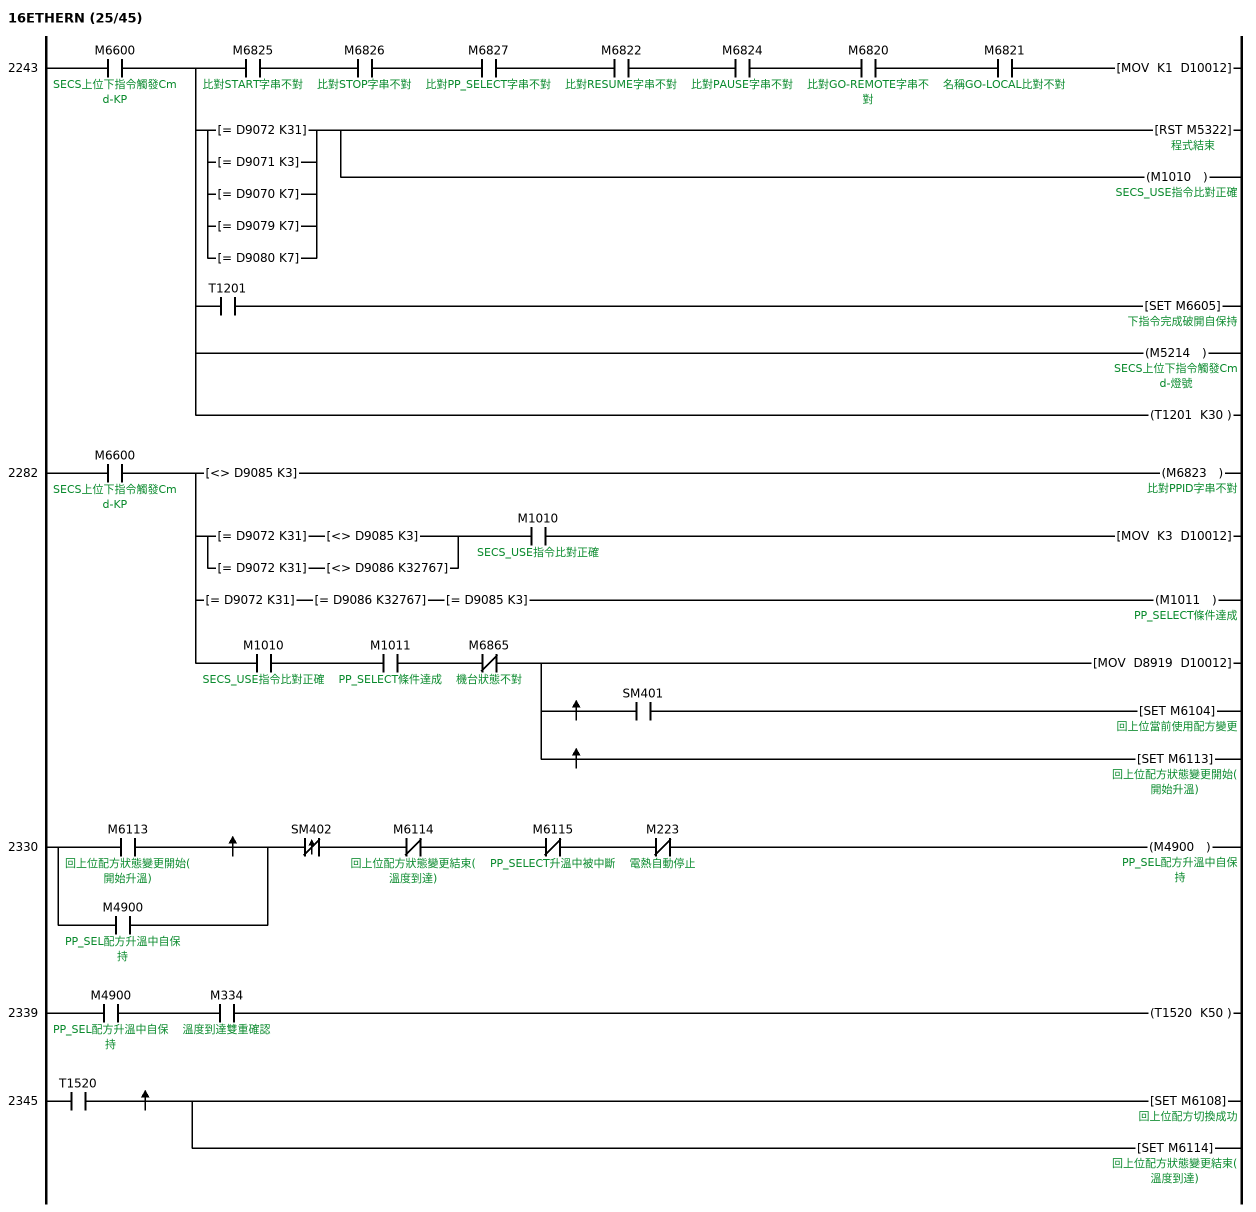
[picture p120: ladder of 16ETHERN, rungs at steps 2243 to 2345]
2243  LD      M6600  ; SECS上位下指令觸發Cmd-KP
      MPS
      AND     M6825  ; 比對START字串不對
      AND     M6826  ; 比對STOP字串不對
      AND     M6827  ; 比對PP_SELECT字串不對
      AND     M6822  ; 比對RESUME字串不對
      AND     M6824  ; 比對PAUSE字串不對
      AND     M6820  ; 比對GO-REMOTE字串不對
      AND     M6821  ; 名稱GO-LOCAL比對不對
      MOV     K1 D10012
      MRD
      LD=     D9072 K31
      OR=     D9071 K3
      OR=     D9070 K7
      OR=     D9079 K7
      OR=     D9080 K7
      ANB
      RST     M5322  ; 程式結束
      OUT     M1010  ; SECS_USE指令比對正確
      MRD
      AND     T1201
      SET     M6605  ; 下指令完成破開自保持
      MPP
      OUT     M5214  ; SECS上位下指令觸發Cmd-燈號
      OUT     T1201 K30
2282  LD      M6600  ; SECS上位下指令觸發Cmd-KP
      MPS
      AND<>   D9085 K3
      OUT     M6823  ; 比對PPID字串不對
      MRD
      LD=     D9072 K31
      AND<>   D9085 K3
      LD=     D9072 K31
      AND<>   D9086 K32767
      ORB
      ANB
      AND     M1010  ; SECS_USE指令比對正確
      MOV     K3 D10012
      MRD
      AND=    D9072 K31
      AND=    D9086 K32767
      AND=    D9085 K3
      OUT     M1011  ; PP_SELECT條件達成
      MPP
      AND     M1010  ; SECS_USE指令比對正確
      AND     M1011  ; PP_SELECT條件達成
      ANI     M6865  ; 機台狀態不對
      MOV     D8919 D10012
      MPS
      MEP
      AND     SM401
      SET     M6104  ; 回上位當前使用配方變更
      MPP
      MEP
      SET     M6113  ; 回上位配方狀態變更開始(開始升溫)
2330  LD      M6113  ; 回上位配方狀態變更開始(開始升溫)
      MEP
      OR      M4900  ; PP_SEL配方升溫中自保持
      ANDPI   SM402
      ANI     M6114  ; 回上位配方狀態變更結束(溫度到達)
      ANI     M6115  ; PP_SELECT升溫中被中斷
      ANI     M223  ; 電熱自動停止
      OUT     M4900  ; PP_SEL配方升溫中自保持
2339  LD      M4900  ; PP_SEL配方升溫中自保持
      AND     M334  ; 溫度到達雙重確認
      OUT     T1520 K50
2345  LD      T1520
      MEP
      SET     M6108  ; 回上位配方切換成功
      SET     M6114  ; 回上位配方狀態變更結束(溫度到達)
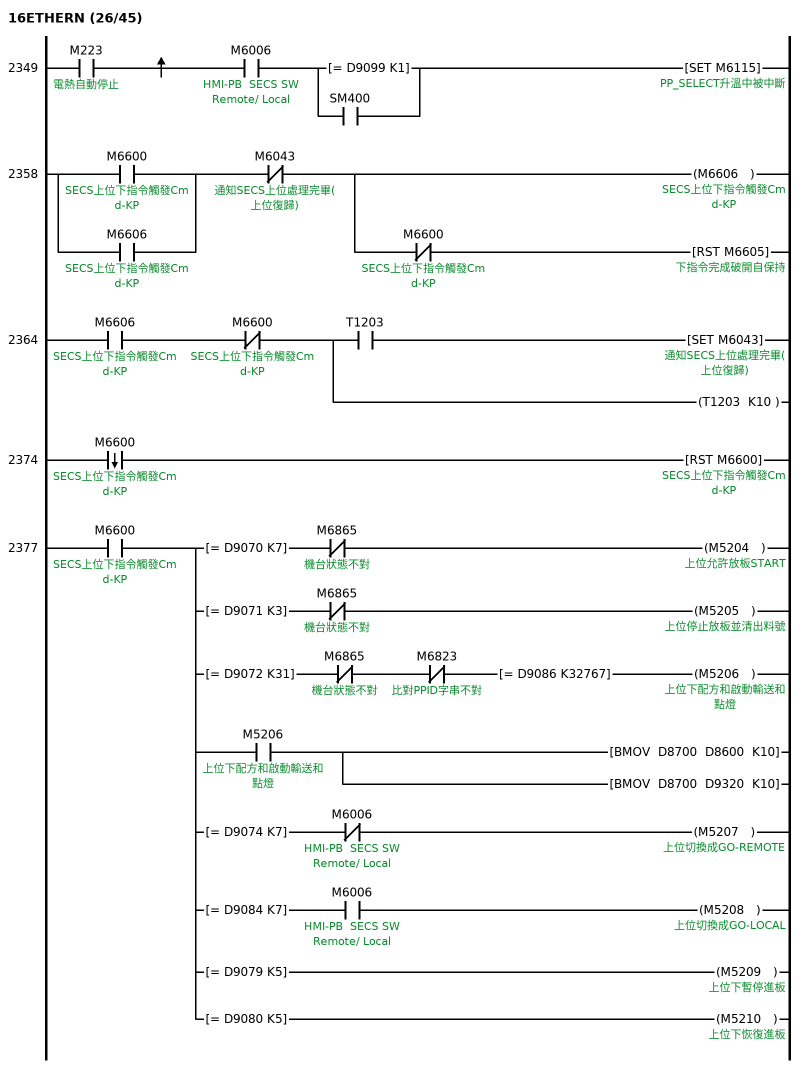
2349  LD      M223  ; 電熱自動停止
      MEP
      AND     M6006  ; HMI-PB  SECS SW  Remote/ Local
      LD=     D9099 K1
      OR      SM400
      ANB
      SET     M6115  ; PP_SELECT升溫中被中斷
2358  LD      M6600  ; SECS上位下指令觸發Cmd-KP
      OR      M6606  ; SECS上位下指令觸發Cmd-KP
      ANI     M6043  ; 通知SECS上位處理完畢(上位復歸)
      OUT     M6606  ; SECS上位下指令觸發Cmd-KP
      ANI     M6600  ; SECS上位下指令觸發Cmd-KP
      RST     M6605  ; 下指令完成破開自保持
2364  LD      M6606  ; SECS上位下指令觸發Cmd-KP
      ANI     M6600  ; SECS上位下指令觸發Cmd-KP
      MPS
      AND     T1203
      SET     M6043  ; 通知SECS上位處理完畢(上位復歸)
      MPP
      OUT     T1203 K10
2374  LDF     M6600  ; SECS上位下指令觸發Cmd-KP
      RST     M6600  ; SECS上位下指令觸發Cmd-KP
2377  LD      M6600  ; SECS上位下指令觸發Cmd-KP
      MPS
      AND=    D9070 K7
      ANI     M6865  ; 機台狀態不對
      OUT     M5204  ; 上位允許放板START
      MRD
      AND=    D9071 K3
      ANI     M6865  ; 機台狀態不對
      OUT     M5205  ; 上位停止放板並清出料號
      MRD
      AND=    D9072 K31
      ANI     M6865  ; 機台狀態不對
      ANI     M6823  ; 比對PPID字串不對
      AND=    D9086 K32767
      OUT     M5206  ; 上位下配方和啟動輸送和點燈
      MRD
      AND     M5206  ; 上位下配方和啟動輸送和點燈
      BMOV    D8700 D8600 K10
      BMOV    D8700 D9320 K10
      MRD
      AND=    D9074 K7
      ANI     M6006  ; HMI-PB  SECS SW  Remote/ Local
      OUT     M5207  ; 上位切換成GO-REMOTE
      MRD
      AND=    D9084 K7
      AND     M6006  ; HMI-PB  SECS SW  Remote/ Local
      OUT     M5208  ; 上位切換成GO-LOCAL
      MRD
      AND=    D9079 K5
      OUT     M5209  ; 上位下暫停進板
      MPP
      AND=    D9080 K5
      OUT     M5210  ; 上位下恢復進板
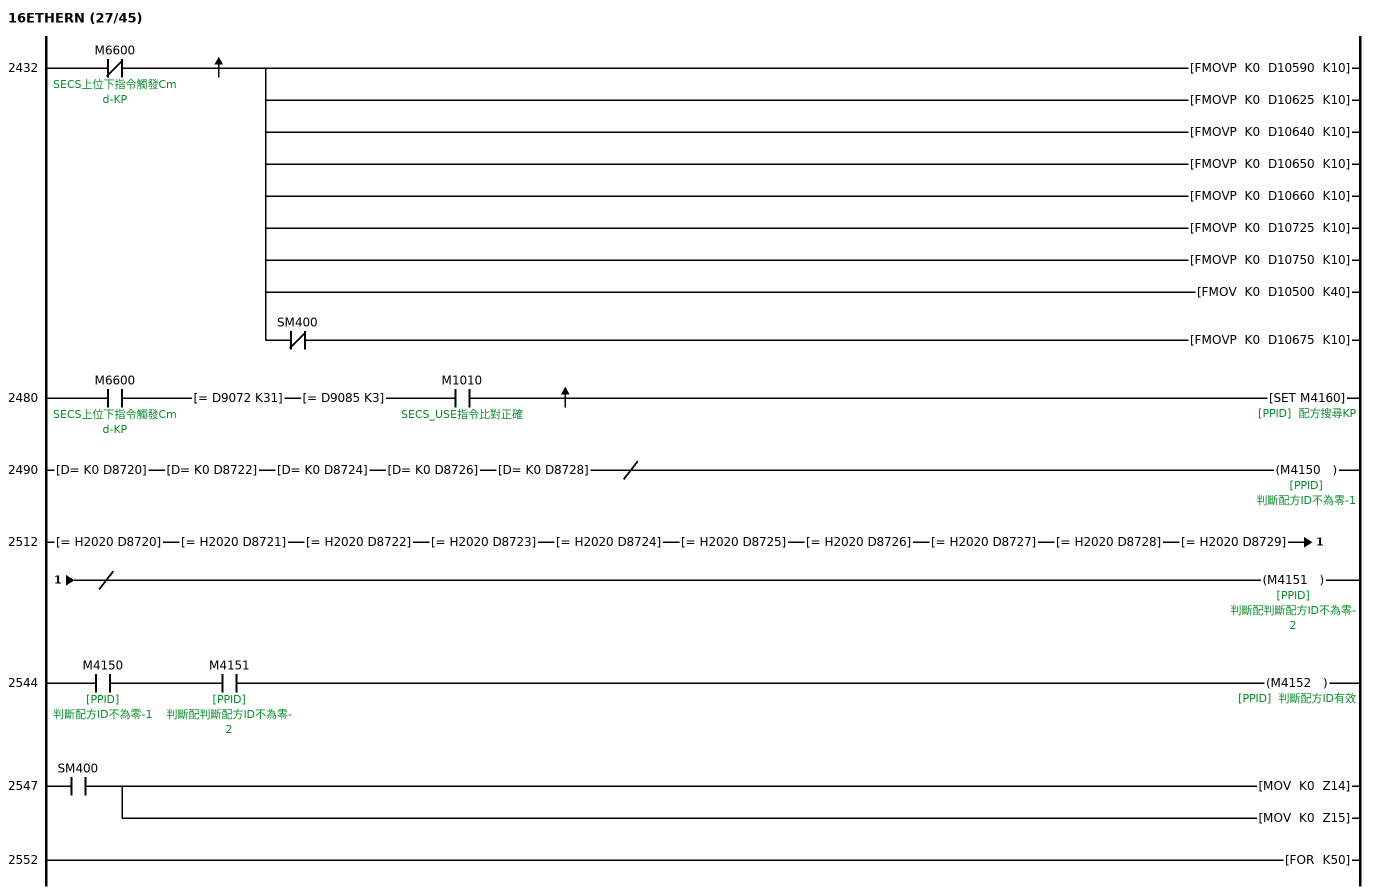
2432  LDI     M6600  ; SECS上位下指令觸發Cmd-KP
      MEP
      FMOVP   K0 D10590 K10
      FMOVP   K0 D10625 K10
      FMOVP   K0 D10640 K10
      FMOVP   K0 D10650 K10
      FMOVP   K0 D10660 K10
      FMOVP   K0 D10725 K10
      FMOVP   K0 D10750 K10
      FMOV    K0 D10500 K40
      ANI     SM400
      FMOVP   K0 D10675 K10
2480  LD      M6600  ; SECS上位下指令觸發Cmd-KP
      AND=    D9072 K31
      AND=    D9085 K3
      AND     M1010  ; SECS_USE指令比對正確
      MEP
      SET     M4160  ; [PPID]  配方搜尋KP
2490  LDD=    K0 D8720
      ANDD=   K0 D8722
      ANDD=   K0 D8724
      ANDD=   K0 D8726
      ANDD=   K0 D8728
      INV
      OUT     M4150  ; [PPID]  判斷配方ID不為零-1
2512  LD=     H2020 D8720
      AND=    H2020 D8721
      AND=    H2020 D8722
      AND=    H2020 D8723
      AND=    H2020 D8724
      AND=    H2020 D8725
      AND=    H2020 D8726
      AND=    H2020 D8727
      AND=    H2020 D8728
      AND=    H2020 D8729
      INV
      OUT     M4151  ; [PPID]  判斷配判斷配方ID不為零-2
2544  LD      M4150  ; [PPID]  判斷配方ID不為零-1
      AND     M4151  ; [PPID]  判斷配判斷配方ID不為零-2
      OUT     M4152  ; [PPID]  判斷配方ID有效
2547  LD      SM400
      MOV     K0 Z14
      MOV     K0 Z15
2552  FOR     K50
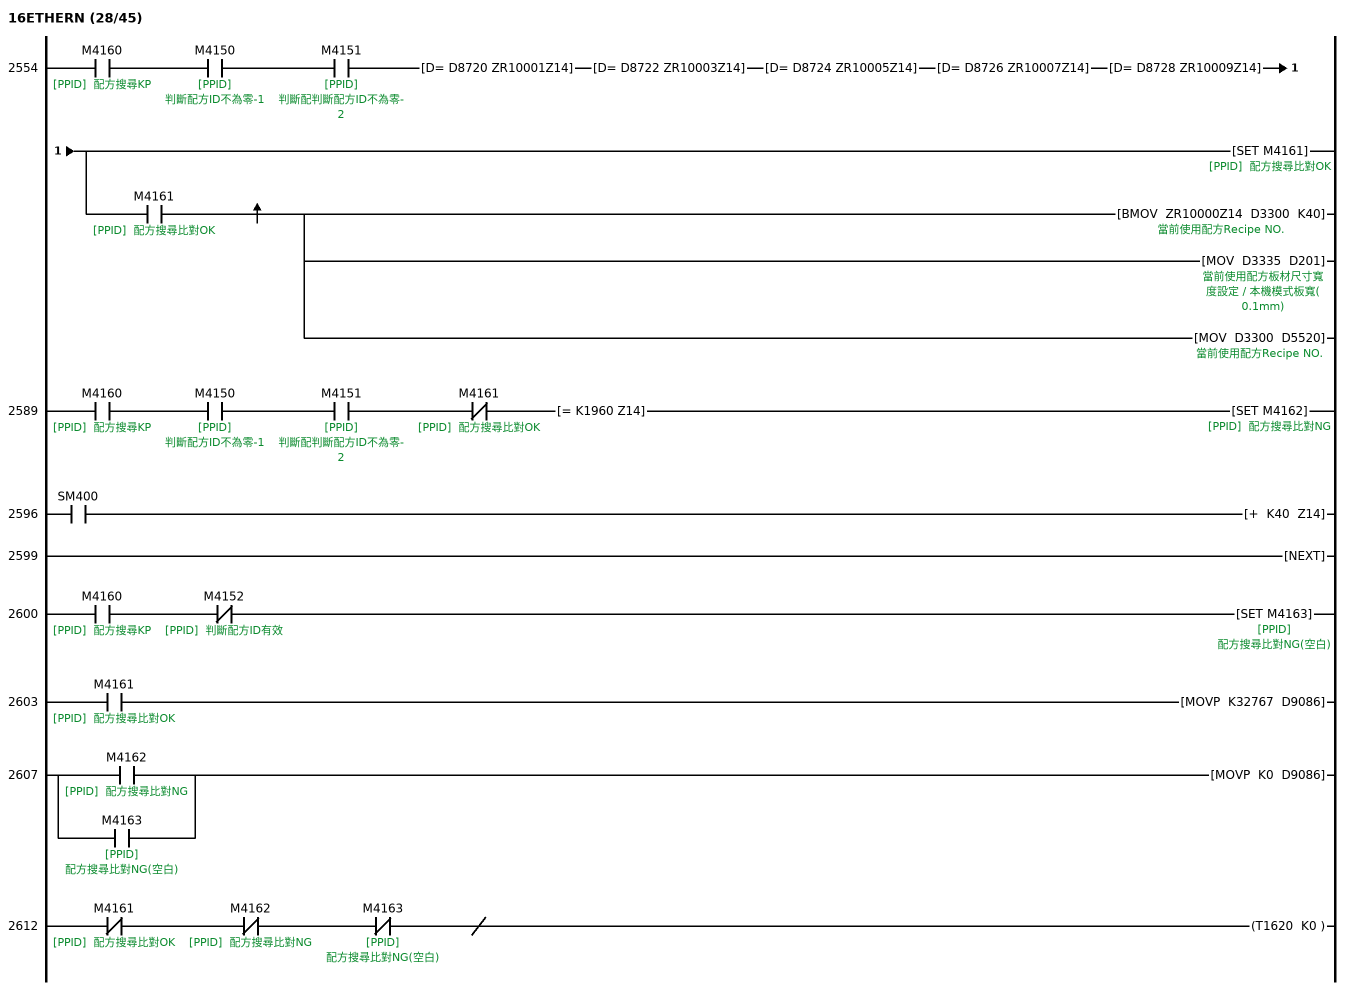
2554  LD      M4160  ; [PPID]  配方搜尋KP
      AND     M4150  ; [PPID]  判斷配方ID不為零-1
      AND     M4151  ; [PPID]  判斷配判斷配方ID不為零-2
      ANDD=   D8720 ZR10001Z14
      ANDD=   D8722 ZR10003Z14
      ANDD=   D8724 ZR10005Z14
      ANDD=   D8726 ZR10007Z14
      ANDD=   D8728 ZR10009Z14
      SET     M4161  ; [PPID]  配方搜尋比對OK
      AND     M4161  ; [PPID]  配方搜尋比對OK
      MEP
      BMOV    ZR10000Z14 D3300 K40  ; 當前使用配方Recipe NO.
      MOV     D3335 D201  ; 當前使用配方板材尺寸寬度設定 / 本機模式板寬(0.1mm)
      MOV     D3300 D5520
2589  LD      M4160  ; [PPID]  配方搜尋KP
      AND     M4150  ; [PPID]  判斷配方ID不為零-1
      AND     M4151  ; [PPID]  判斷配判斷配方ID不為零-2
      ANI     M4161  ; [PPID]  配方搜尋比對OK
      AND=    K1960 Z14
      SET     M4162  ; [PPID]  配方搜尋比對NG
2596  LD      SM400
      +       K40 Z14
2599  NEXT
2600  LD      M4160  ; [PPID]  配方搜尋KP
      ANI     M4152  ; [PPID]  判斷配方ID有效
      SET     M4163  ; [PPID]  配方搜尋比對NG(空白)
2603  LD      M4161  ; [PPID]  配方搜尋比對OK
      MOVP    K32767 D9086
2607  LD      M4162  ; [PPID]  配方搜尋比對NG
      OR      M4163  ; [PPID]  配方搜尋比對NG(空白)
      MOVP    K0 D9086
2612  LDI     M4161  ; [PPID]  配方搜尋比對OK
      ANI     M4162  ; [PPID]  配方搜尋比對NG
      ANI     M4163  ; [PPID]  配方搜尋比對NG(空白)
      INV
      OUT     T1620 K0
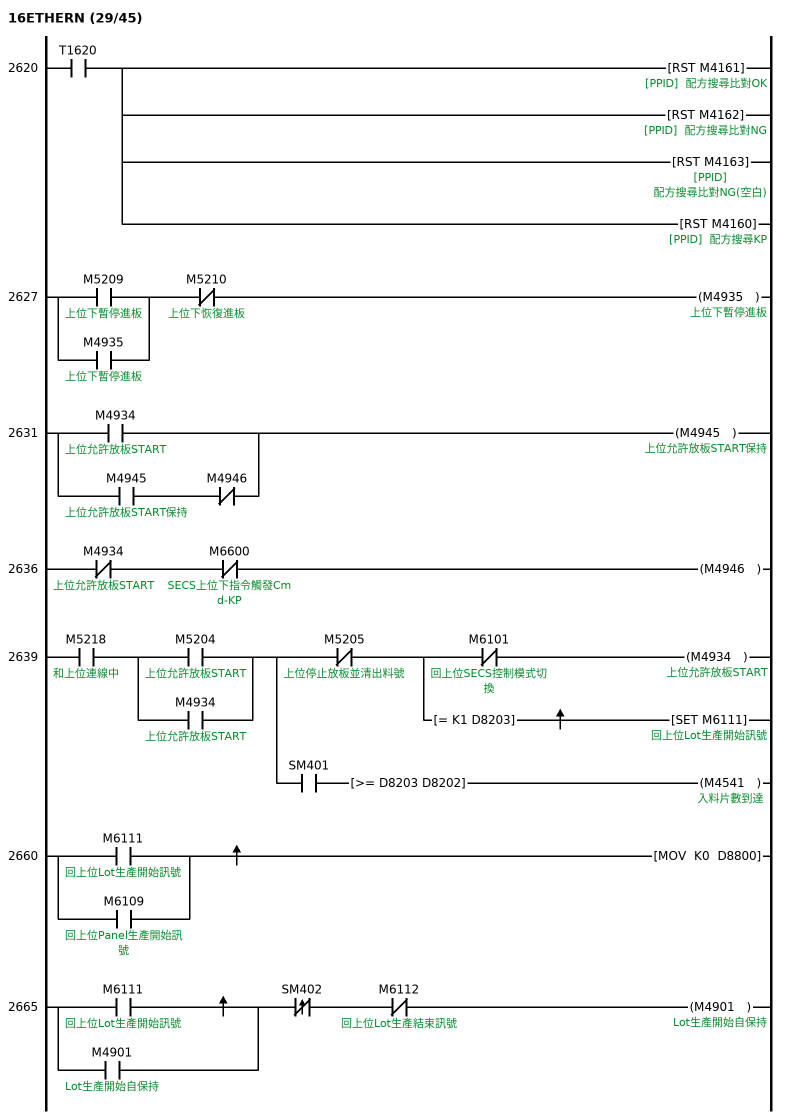
2620  LD      T1620
      RST     M4161  ; [PPID]  配方搜尋比對OK
      RST     M4162  ; [PPID]  配方搜尋比對NG
      RST     M4163  ; [PPID]  配方搜尋比對NG(空白)
      RST     M4160  ; [PPID]  配方搜尋KP
2627  LD      M5209  ; 上位下暫停進板
      OR      M4935  ; 上位下暫停進板
      ANI     M5210  ; 上位下恢復進板
      OUT     M4935  ; 上位下暫停進板
2631  LD      M4934  ; 上位允許放板START
      LD      M4945  ; 上位允許放板START保持
      ANI     M4946
      ORB
      OUT     M4945  ; 上位允許放板START保持
2636  LDI     M4934  ; 上位允許放板START
      ANI     M6600  ; SECS上位下指令觸發Cmd-KP
      OUT     M4946
2639  LD      M5218  ; 和上位連線中
      LD      M5204  ; 上位允許放板START
      OR      M4934  ; 上位允許放板START
      ANB
      MPS
      ANI     M5205  ; 上位停止放板並清出料號
      MPS
      ANI     M6101  ; 回上位SECS控制模式切換
      OUT     M4934  ; 上位允許放板START
      MPP
      AND=    K1 D8203
      MEP
      SET     M6111  ; 回上位Lot生產開始訊號
      MPP
      AND     SM401
      AND>=   D8203 D8202
      OUT     M4541  ; 入料片數到達
2660  LD      M6111  ; 回上位Lot生產開始訊號
      OR      M6109  ; 回上位Panel生產開始訊號
      MEP
      MOV     K0 D8800
2665  LD      M6111  ; 回上位Lot生產開始訊號
      MEP
      OR      M4901  ; Lot生產開始自保持
      ANDPI   SM402
      ANI     M6112  ; 回上位Lot生產結束訊號
      OUT     M4901  ; Lot生產開始自保持
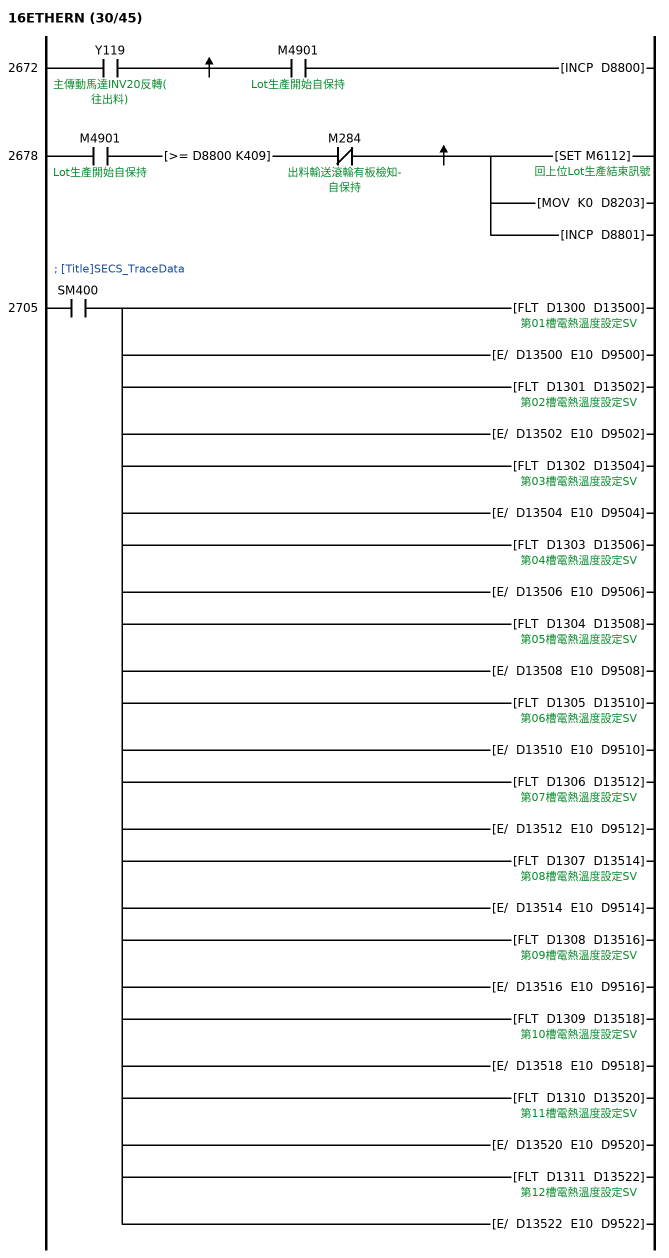
2672  LD      Y119  ; 主傳動馬達INV20反轉(往出料)
      MEP
      AND     M4901  ; Lot生產開始自保持
      INCP    D8800
2678  LD      M4901  ; Lot生產開始自保持
      AND>=   D8800 K409
      ANI     M284  ; 出料輸送滾輪有板檢知-自保持
      MEP
      SET     M6112  ; 回上位Lot生產結束訊號
      MOV     K0 D8203
      INCP    D8801
; [Title]SECS_TraceData
2705  LD      SM400
      FLT     D1300 D13500  ; 第01槽電熱溫度設定SV
      E/      D13500 E10 D9500
      FLT     D1301 D13502  ; 第02槽電熱溫度設定SV
      E/      D13502 E10 D9502
      FLT     D1302 D13504  ; 第03槽電熱溫度設定SV
      E/      D13504 E10 D9504
      FLT     D1303 D13506  ; 第04槽電熱溫度設定SV
      E/      D13506 E10 D9506
      FLT     D1304 D13508  ; 第05槽電熱溫度設定SV
      E/      D13508 E10 D9508
      FLT     D1305 D13510  ; 第06槽電熱溫度設定SV
      E/      D13510 E10 D9510
      FLT     D1306 D13512  ; 第07槽電熱溫度設定SV
      E/      D13512 E10 D9512
      FLT     D1307 D13514  ; 第08槽電熱溫度設定SV
      E/      D13514 E10 D9514
      FLT     D1308 D13516  ; 第09槽電熱溫度設定SV
      E/      D13516 E10 D9516
      FLT     D1309 D13518  ; 第10槽電熱溫度設定SV
      E/      D13518 E10 D9518
      FLT     D1310 D13520  ; 第11槽電熱溫度設定SV
      E/      D13520 E10 D9520
      FLT     D1311 D13522  ; 第12槽電熱溫度設定SV
      E/      D13522 E10 D9522
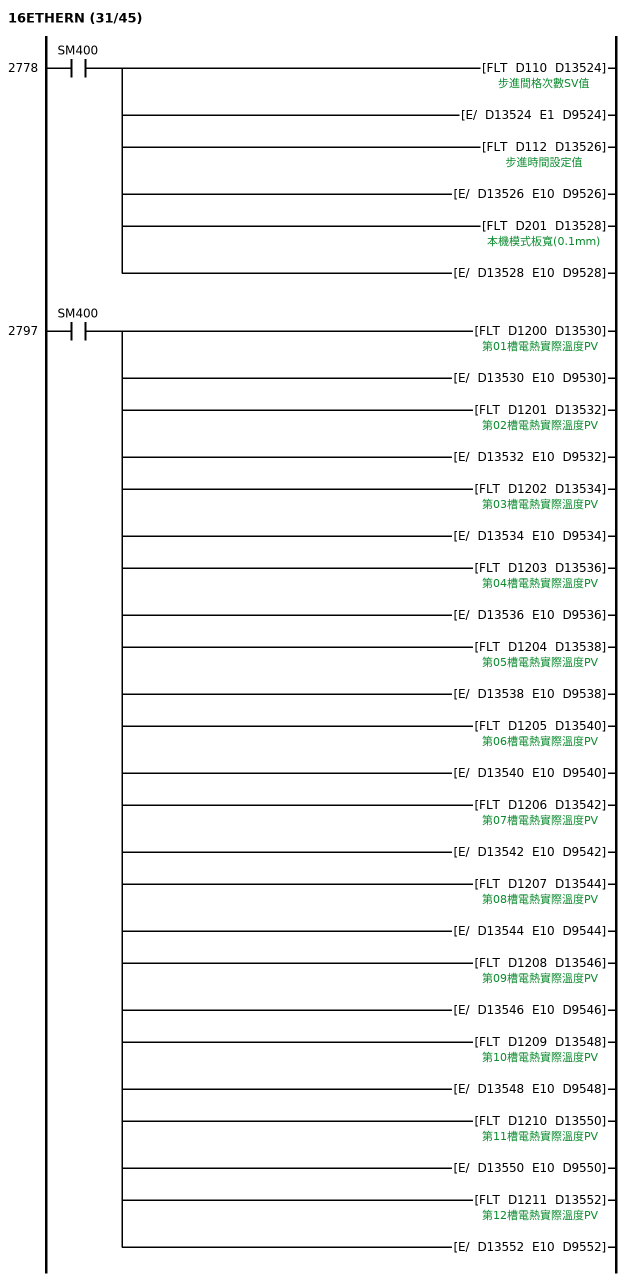
2778  LD      SM400
      FLT     D110 D13524  ; 步進間格次數SV值
      E/      D13524 E1 D9524
      FLT     D112 D13526  ; 步進時間設定值
      E/      D13526 E10 D9526
      FLT     D201 D13528
      E/      D13528 E10 D9528
2797  LD      SM400
      FLT     D1200 D13530
      E/      D13530 E10 D9530
      FLT     D1201 D13532
      E/      D13532 E10 D9532
      FLT     D1202 D13534
      E/      D13534 E10 D9534
      FLT     D1203 D13536
      E/      D13536 E10 D9536
      FLT     D1204 D13538
      E/      D13538 E10 D9538
      FLT     D1205 D13540
      E/      D13540 E10 D9540
      FLT     D1206 D13542
      E/      D13542 E10 D9542
      FLT     D1207 D13544
      E/      D13544 E10 D9544
      FLT     D1208 D13546
      E/      D13546 E10 D9546
      FLT     D1209 D13548
      E/      D13548 E10 D9548
      FLT     D1210 D13550
      E/      D13550 E10 D9550
      FLT     D1211 D13552
      E/      D13552 E10 D9552
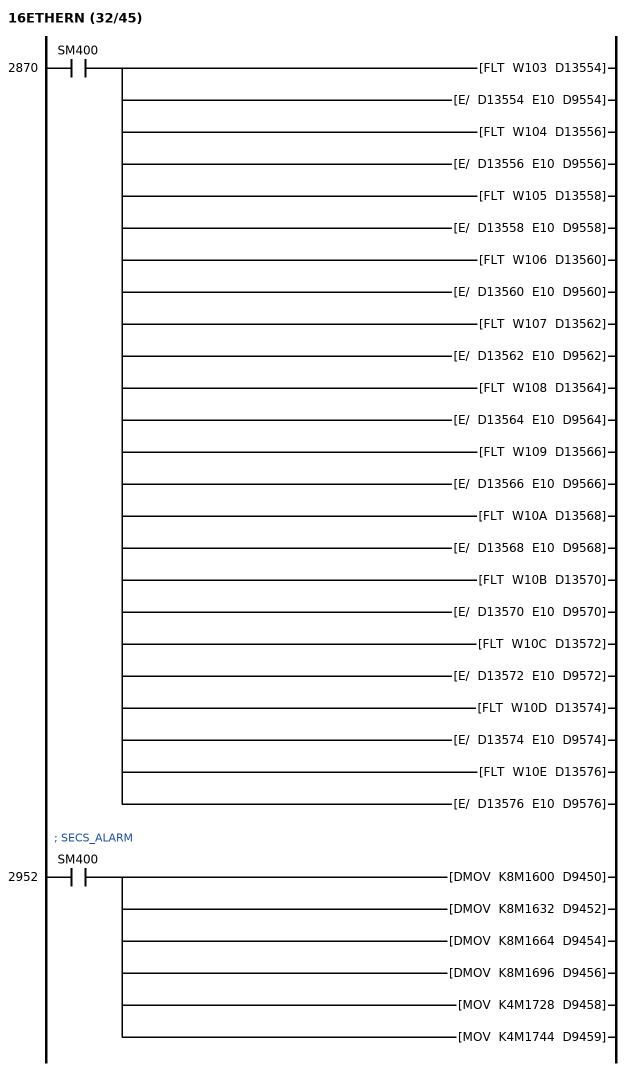
2870  LD      SM400
      FLT     W103 D13554
      E/      D13554 E10 D9554
      FLT     W104 D13556
      E/      D13556 E10 D9556
      FLT     W105 D13558
      E/      D13558 E10 D9558
      FLT     W106 D13560
      E/      D13560 E10 D9560
      FLT     W107 D13562
      E/      D13562 E10 D9562
      FLT     W108 D13564
      E/      D13564 E10 D9564
      FLT     W109 D13566
      E/      D13566 E10 D9566
      FLT     W10A D13568
      E/      D13568 E10 D9568
      FLT     W10B D13570
      E/      D13570 E10 D9570
      FLT     W10C D13572
      E/      D13572 E10 D9572
      FLT     W10D D13574
      E/      D13574 E10 D9574
      FLT     W10E D13576
      E/      D13576 E10 D9576
; SECS_ALARM
2952  LD      SM400
      DMOV    K8M1600 D9450
      DMOV    K8M1632 D9452
      DMOV    K8M1664 D9454  ; 出料風車1過載異常
      DMOV    K8M1696 D9456  ; 進料夾爪開異常
      MOV     K4M1728 D9458  ; 緊急停止異常
      MOV     K4M1744 D9459  ; #01分路開關跳脫
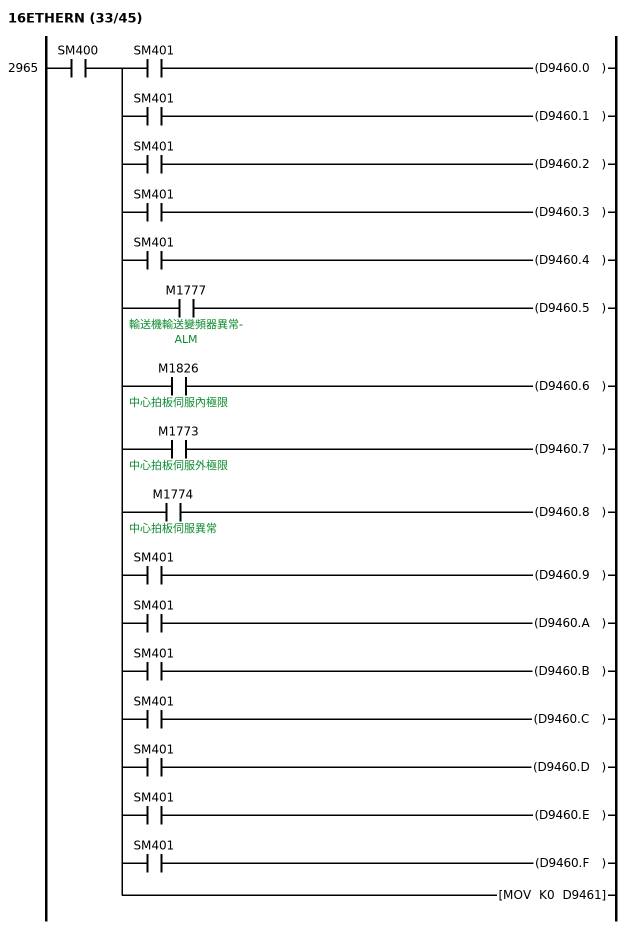
2965  LD      SM400
      MPS
      AND     SM401
      OUT     D9460.0
      MRD
      AND     SM401
      OUT     D9460.1
      MRD
      AND     SM401
      OUT     D9460.2
      MRD
      AND     SM401
      OUT     D9460.3
      MRD
      AND     SM401
      OUT     D9460.4
      MRD
      AND     M1777  ; 輸送機輸送變頻器異常-ALM
      OUT     D9460.5
      MRD
      AND     M1826  ; 中心拍板伺服內極限
      OUT     D9460.6
      MRD
      AND     M1773  ; 中心拍板伺服外極限
      OUT     D9460.7
      MRD
      AND     M1774  ; 中心拍板伺服異常
      OUT     D9460.8
      MRD
      AND     SM401
      OUT     D9460.9
      MRD
      AND     SM401
      OUT     D9460.A
      MRD
      AND     SM401
      OUT     D9460.B
      MRD
      AND     SM401
      OUT     D9460.C
      MRD
      AND     SM401
      OUT     D9460.D
      MRD
      AND     SM401
      OUT     D9460.E
      MRD
      AND     SM401
      OUT     D9460.F
      MPP
      MOV     K0 D9461
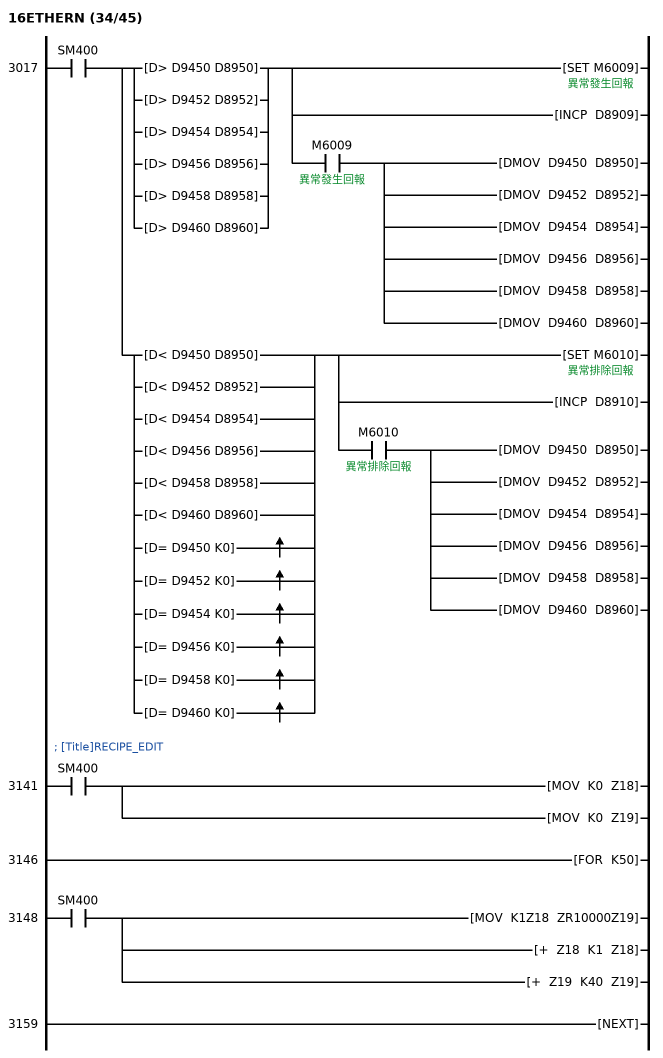
3017  LD      SM400
      MPS
      LDD>    D9450 D8950
      ORD>    D9452 D8952
      ORD>    D9454 D8954
      ORD>    D9456 D8956
      ORD>    D9458 D8958
      ORD>    D9460 D8960
      ANB
      SET     M6009  ; 異常發生回報
      INCP    D8909
      AND     M6009  ; 異常發生回報
      DMOV    D9450 D8950
      DMOV    D9452 D8952
      DMOV    D9454 D8954
      DMOV    D9456 D8956
      DMOV    D9458 D8958
      DMOV    D9460 D8960
      MPP
      LDD<    D9450 D8950
      ORD<    D9452 D8952
      ORD<    D9454 D8954
      ORD<    D9456 D8956
      ORD<    D9458 D8958
      ORD<    D9460 D8960
      LDD=    D9450 K0
      MEP
      ORB
      LDD=    D9452 K0
      MEP
      ORB
      LDD=    D9454 K0
      MEP
      ORB
      LDD=    D9456 K0
      MEP
      ORB
      LDD=    D9458 K0
      MEP
      ORB
      LDD=    D9460 K0
      MEP
      ORB
      ANB
      SET     M6010  ; 異常排除回報
      INCP    D8910
      AND     M6010  ; 異常排除回報
      DMOV    D9450 D8950
      DMOV    D9452 D8952
      DMOV    D9454 D8954
      DMOV    D9456 D8956
      DMOV    D9458 D8958
      DMOV    D9460 D8960
; [Title]RECIPE_EDIT
3141  LD      SM400
      MOV     K0 Z18
      MOV     K0 Z19
3146  FOR     K50
3148  LD      SM400
      MOV     K1Z18 ZR10000Z19
      +       Z18 K1 Z18
      +       Z19 K40 Z19
3159  NEXT
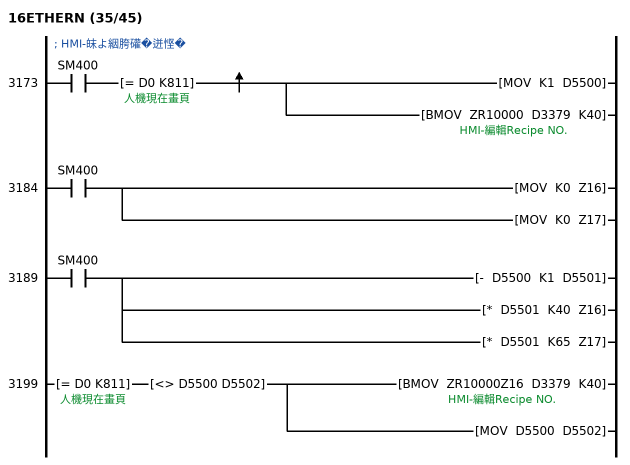
; HMI-配方編輯畫面顯示
3173  LD      SM400
      AND=    D0 K811  ; 人機現在畫頁
      MEP
      MOV     K1 D5500
      BMOV    ZR10000 D3379 K40  ; HMI-編輯Recipe NO.
3184  LD      SM400
      MOV     K0 Z16
      MOV     K0 Z17
3189  LD      SM400
      -       D5500 K1 D5501
      *       D5501 K40 Z16
      *       D5501 K65 Z17
3199  LD=     D0 K811  ; 人機現在畫頁
      AND<>   D5500 D5502
      BMOV    ZR10000Z16 D3379 K40
      MOV     D5500 D5502
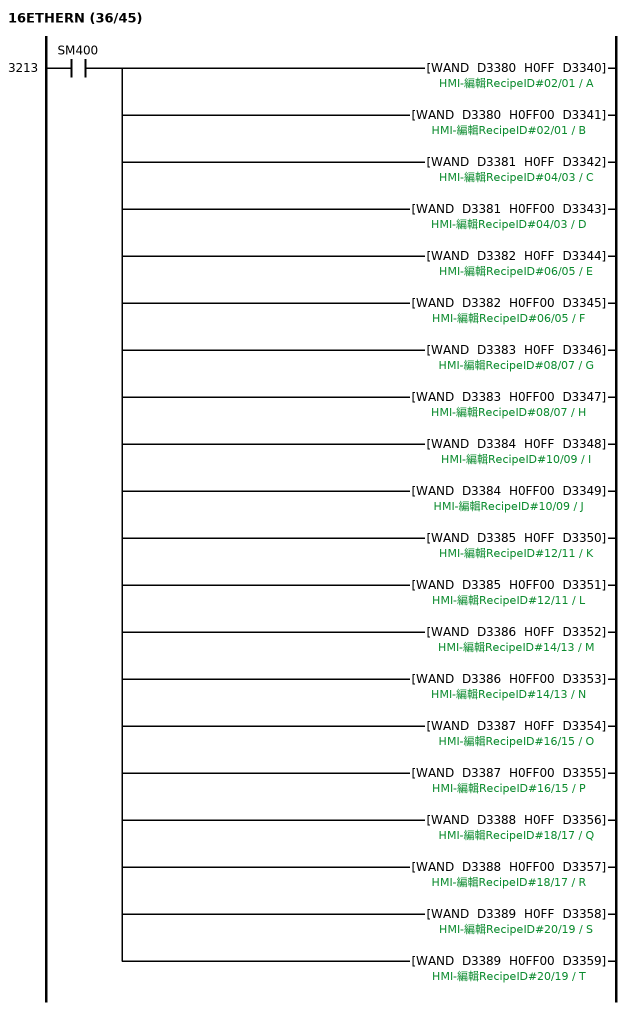
3213  LD      SM400
      WAND    D3380 H0FF D3340  ; HMI-編輯RecipeID#02/01 / A
      WAND    D3380 H0FF00 D3341  ; B
      WAND    D3381 H0FF D3342  ; HMI-編輯RecipeID#04/03 / C
      WAND    D3381 H0FF00 D3343  ; D
      WAND    D3382 H0FF D3344  ; HMI-編輯RecipeID#06/05 / E
      WAND    D3382 H0FF00 D3345  ; F
      WAND    D3383 H0FF D3346  ; HMI-編輯RecipeID#08/07 / G
      WAND    D3383 H0FF00 D3347  ; H
      WAND    D3384 H0FF D3348  ; HMI-編輯RecipeID#10/09 / I
      WAND    D3384 H0FF00 D3349  ; J
      WAND    D3385 H0FF D3350  ; HMI-編輯RecipeID#12/11 / K
      WAND    D3385 H0FF00 D3351  ; L
      WAND    D3386 H0FF D3352  ; HMI-編輯RecipeID#14/13 / M
      WAND    D3386 H0FF00 D3353  ; N
      WAND    D3387 H0FF D3354  ; HMI-編輯RecipeID#16/15 / O
      WAND    D3387 H0FF00 D3355  ; P
      WAND    D3388 H0FF D3356  ; HMI-編輯RecipeID#18/17 / Q
      WAND    D3388 H0FF00 D3357  ; R
      WAND    D3389 H0FF D3358  ; HMI-編輯RecipeID#20/19 / S
      WAND    D3389 H0FF00 D3359  ; T
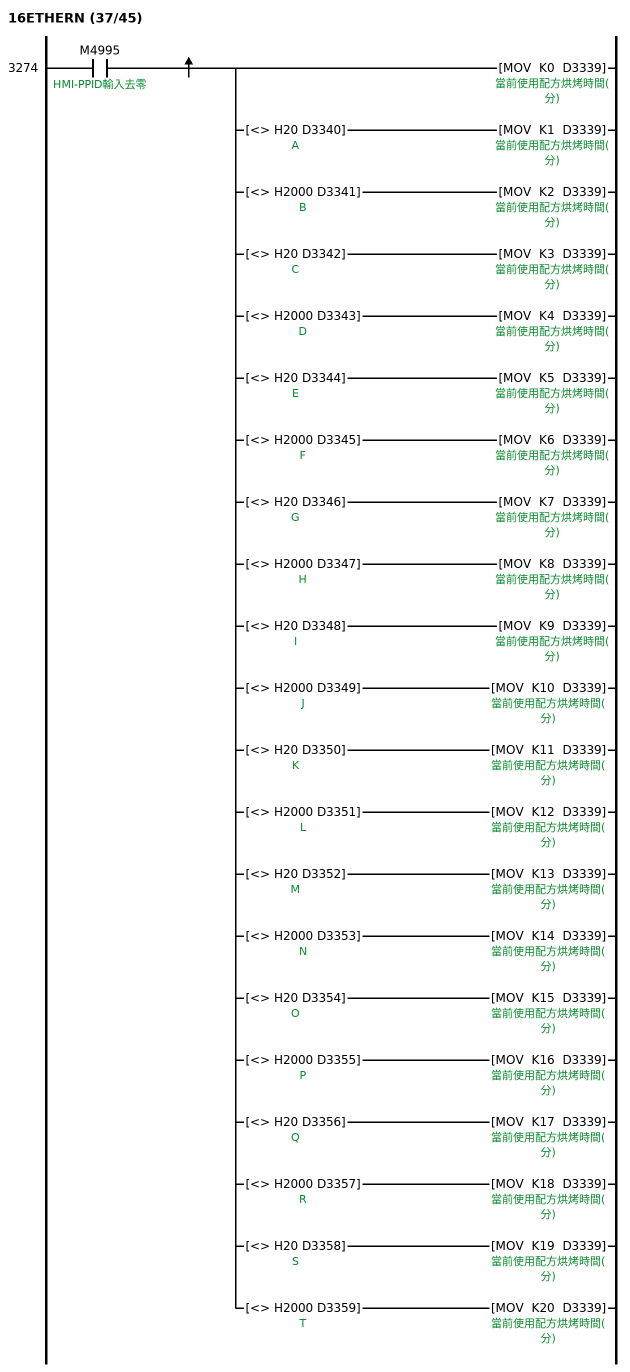
3274  LD      M4995  ; HMI-PPID輸入去零
      MEP
      MOV     K0 D3339  ; 當前使用配方烘烤時間(分)
      MPS
      AND<>   H20 D3340  ; A
      MOV     K1 D3339
      MRD
      AND<>   H2000 D3341  ; B
      MOV     K2 D3339
      MRD
      AND<>   H20 D3342  ; C
      MOV     K3 D3339
      MRD
      AND<>   H2000 D3343  ; D
      MOV     K4 D3339
      MRD
      AND<>   H20 D3344  ; E
      MOV     K5 D3339
      MRD
      AND<>   H2000 D3345  ; F
      MOV     K6 D3339
      MRD
      AND<>   H20 D3346  ; G
      MOV     K7 D3339
      MRD
      AND<>   H2000 D3347  ; H
      MOV     K8 D3339
      MRD
      AND<>   H20 D3348  ; I
      MOV     K9 D3339
      MRD
      AND<>   H2000 D3349  ; J
      MOV     K10 D3339
      MRD
      AND<>   H20 D3350  ; K
      MOV     K11 D3339
      MRD
      AND<>   H2000 D3351  ; L
      MOV     K12 D3339
      MRD
      AND<>   H20 D3352  ; M
      MOV     K13 D3339
      MRD
      AND<>   H2000 D3353  ; N
      MOV     K14 D3339
      MRD
      AND<>   H20 D3354  ; O
      MOV     K15 D3339
      MRD
      AND<>   H2000 D3355  ; P
      MOV     K16 D3339
      MRD
      AND<>   H20 D3356  ; Q
      MOV     K17 D3339
      MRD
      AND<>   H2000 D3357  ; R
      MOV     K18 D3339
      MRD
      AND<>   H20 D3358  ; S
      MOV     K19 D3339
      MPP
      AND<>   H2000 D3359  ; T
      MOV     K20 D3339
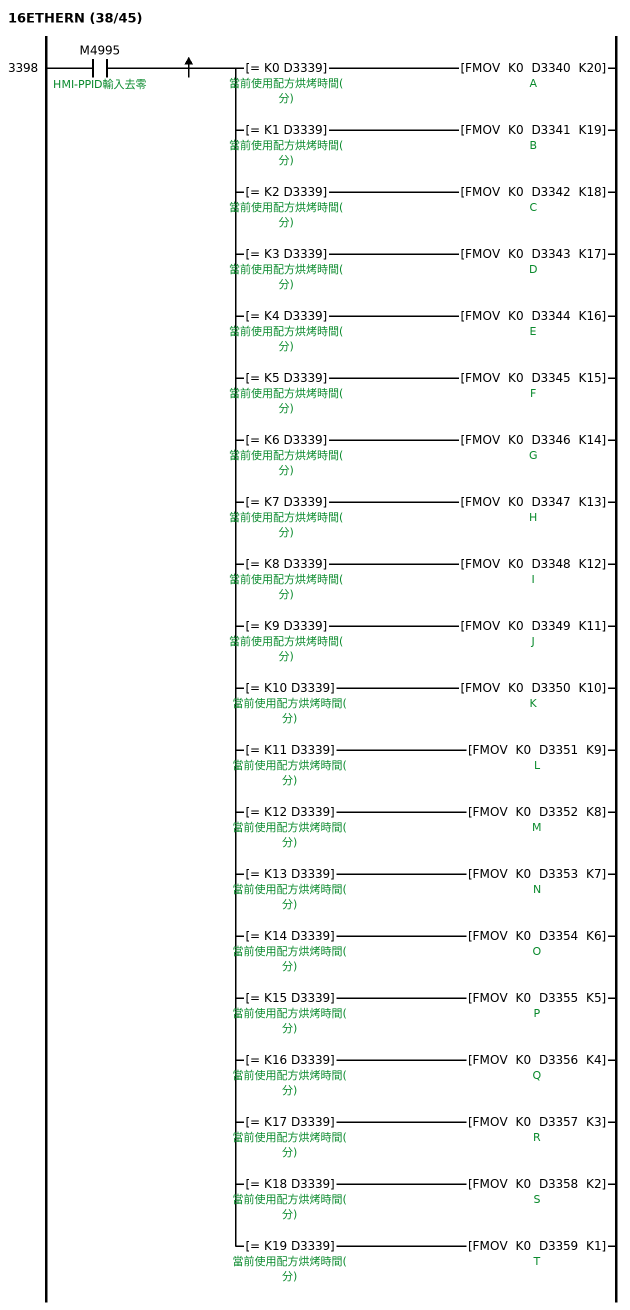
3398  LD      M4995  ; HMI-PPID輸入去零
      MEP
      MPS
      AND=    K0 D3339  ; 當前使用配方烘烤時間(分)
      FMOV    K0 D3340 K20
      MRD
      AND=    K1 D3339  ; 當前使用配方烘烤時間(分)
      FMOV    K0 D3341 K19
      MRD
      AND=    K2 D3339  ; 當前使用配方烘烤時間(分)
      FMOV    K0 D3342 K18
      MRD
      AND=    K3 D3339  ; 當前使用配方烘烤時間(分)
      FMOV    K0 D3343 K17
      MRD
      AND=    K4 D3339  ; 當前使用配方烘烤時間(分)
      FMOV    K0 D3344 K16
      MRD
      AND=    K5 D3339  ; 當前使用配方烘烤時間(分)
      FMOV    K0 D3345 K15
      MRD
      AND=    K6 D3339  ; 當前使用配方烘烤時間(分)
      FMOV    K0 D3346 K14
      MRD
      AND=    K7 D3339  ; 當前使用配方烘烤時間(分)
      FMOV    K0 D3347 K13
      MRD
      AND=    K8 D3339  ; 當前使用配方烘烤時間(分)
      FMOV    K0 D3348 K12
      MRD
      AND=    K9 D3339  ; 當前使用配方烘烤時間(分)
      FMOV    K0 D3349 K11
      MRD
      AND=    K10 D3339  ; 當前使用配方烘烤時間(分)
      FMOV    K0 D3350 K10
      MRD
      AND=    K11 D3339  ; 當前使用配方烘烤時間(分)
      FMOV    K0 D3351 K9
      MRD
      AND=    K12 D3339  ; 當前使用配方烘烤時間(分)
      FMOV    K0 D3352 K8
      MRD
      AND=    K13 D3339  ; 當前使用配方烘烤時間(分)
      FMOV    K0 D3353 K7
      MRD
      AND=    K14 D3339  ; 當前使用配方烘烤時間(分)
      FMOV    K0 D3354 K6
      MRD
      AND=    K15 D3339  ; 當前使用配方烘烤時間(分)
      FMOV    K0 D3355 K5
      MRD
      AND=    K16 D3339  ; 當前使用配方烘烤時間(分)
      FMOV    K0 D3356 K4
      MRD
      AND=    K17 D3339  ; 當前使用配方烘烤時間(分)
      FMOV    K0 D3357 K3
      MRD
      AND=    K18 D3339  ; 當前使用配方烘烤時間(分)
      FMOV    K0 D3358 K2
      MPP
      AND=    K19 D3339  ; 當前使用配方烘烤時間(分)
      FMOV    K0 D3359 K1
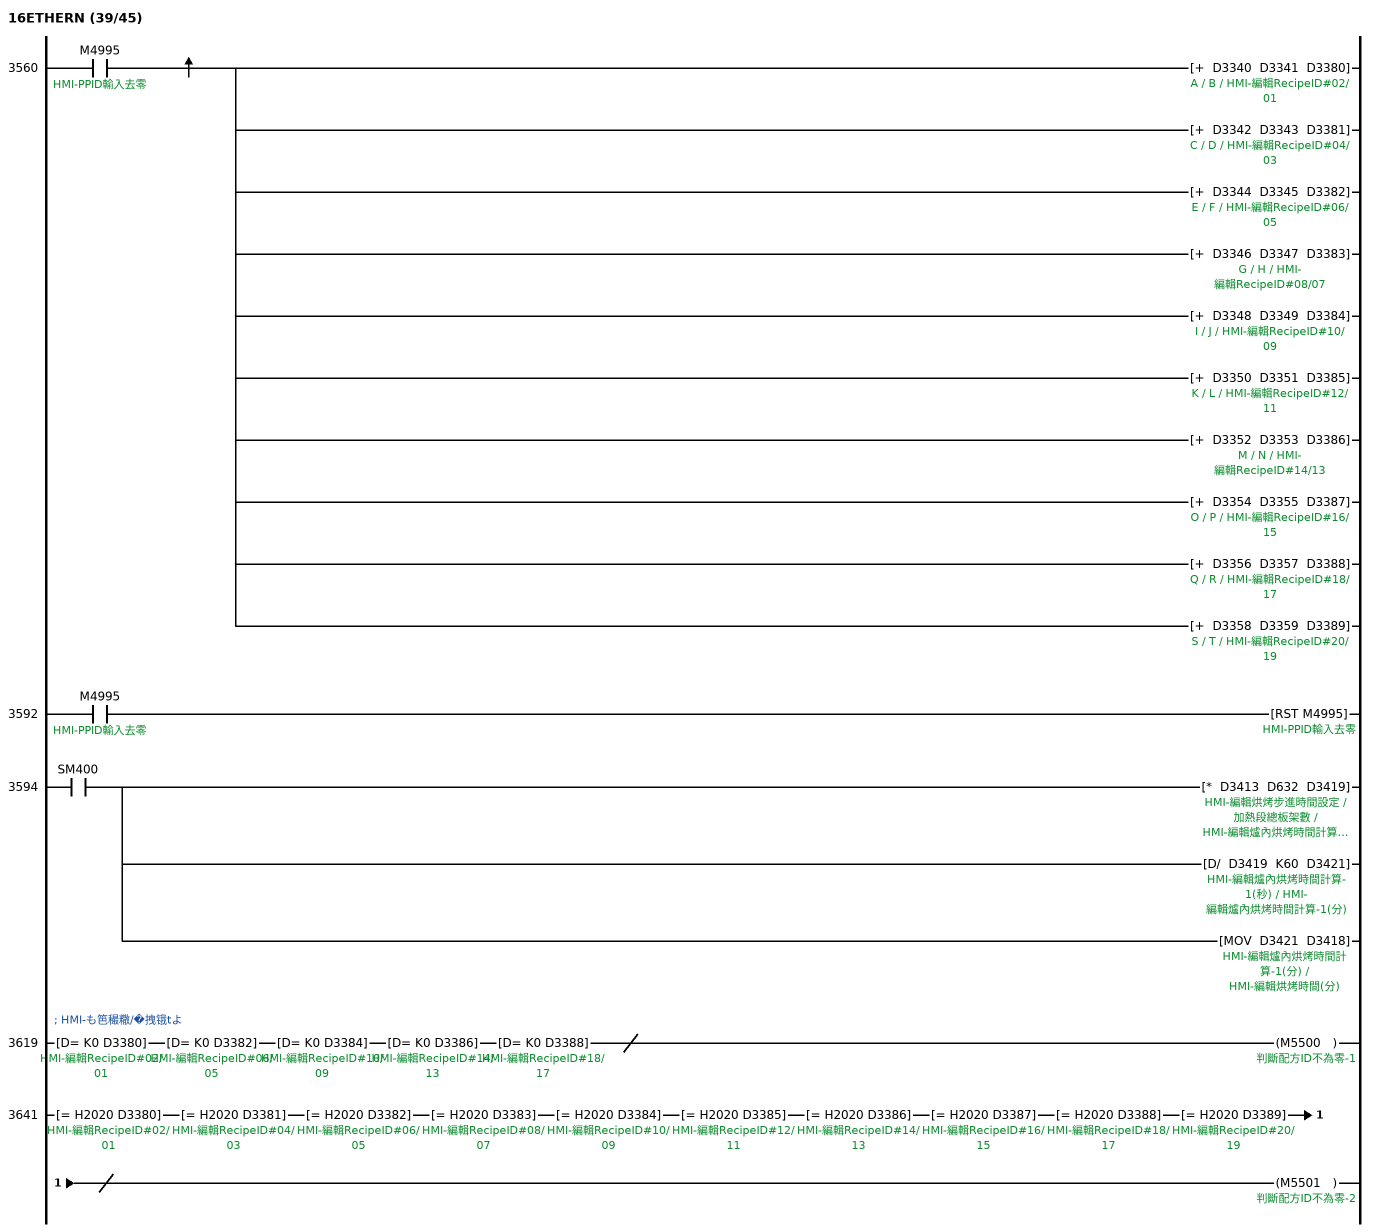
3560  LD      M4995  ; HMI-PPID輸入去零
      MEP
      +       D3340 D3341 D3380
      +       D3342 D3343 D3381
      +       D3344 D3345 D3382
      +       D3346 D3347 D3383
      +       D3348 D3349 D3384
      +       D3350 D3351 D3385
      +       D3352 D3353 D3386
      +       D3354 D3355 D3387
      +       D3356 D3357 D3388
      +       D3358 D3359 D3389
3592  LD      M4995  ; HMI-PPID輸入去零
      RST     M4995  ; HMI-PPID輸入去零
3594  LD      SM400
      *       D3413 D632 D3419  ; HMI-編輯烘烤步進時間設定 / 加熱段總板架數 / HMI-編輯爐內烘烤時間計算-1(秒)
      D/      D3419 K60 D3421  ; HMI-編輯爐內烘烤時間計算-1(分)
      MOV     D3421 D3418  ; HMI-編輯烘烤時間(分)
; HMI-手動新增/修改配方
3619  LDD=    K0 D3380  ; HMI-編輯RecipeID#02/01
      ANDD=   K0 D3382  ; HMI-編輯RecipeID#06/05
      ANDD=   K0 D3384  ; HMI-編輯RecipeID#10/09
      ANDD=   K0 D3386  ; HMI-編輯RecipeID#14/13
      ANDD=   K0 D3388  ; HMI-編輯RecipeID#18/17
      INV
      OUT     M5500  ; 判斷配方ID不為零-1
3641  LD=     H2020 D3380  ; HMI-編輯RecipeID#02/01
      AND=    H2020 D3381  ; HMI-編輯RecipeID#04/03
      AND=    H2020 D3382  ; HMI-編輯RecipeID#06/05
      AND=    H2020 D3383  ; HMI-編輯RecipeID#08/07
      AND=    H2020 D3384  ; HMI-編輯RecipeID#10/09
      AND=    H2020 D3385  ; HMI-編輯RecipeID#12/11
      AND=    H2020 D3386  ; HMI-編輯RecipeID#14/13
      AND=    H2020 D3387  ; HMI-編輯RecipeID#16/15
      AND=    H2020 D3388  ; HMI-編輯RecipeID#18/17
      AND=    H2020 D3389  ; HMI-編輯RecipeID#20/19
      INV
      OUT     M5501  ; 判斷配方ID不為零-2
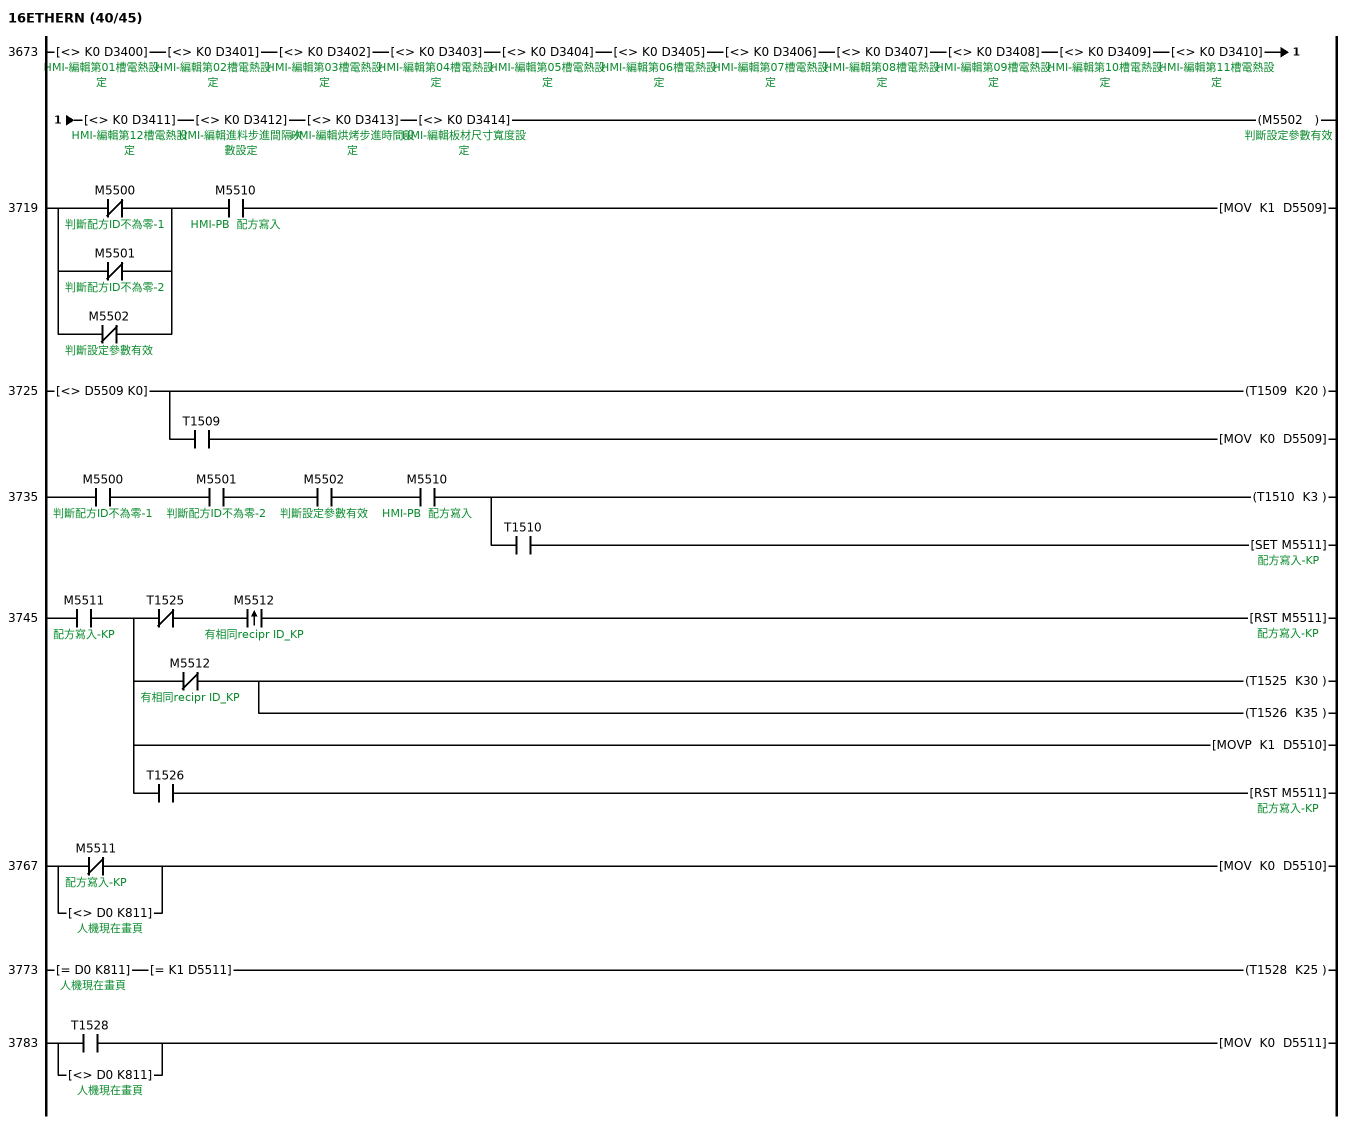
3673  LD<>    K0 D3400  ; HMI-編輯第01槽電熱設定
      AND<>   K0 D3401  ; HMI-編輯第02槽電熱設定
      AND<>   K0 D3402  ; HMI-編輯第03槽電熱設定
      AND<>   K0 D3403  ; HMI-編輯第04槽電熱設定
      AND<>   K0 D3404  ; HMI-編輯第05槽電熱設定
      AND<>   K0 D3405  ; HMI-編輯第06槽電熱設定
      AND<>   K0 D3406  ; HMI-編輯第07槽電熱設定
      AND<>   K0 D3407  ; HMI-編輯第08槽電熱設定
      AND<>   K0 D3408  ; HMI-編輯第09槽電熱設定
      AND<>   K0 D3409  ; HMI-編輯第10槽電熱設定
      AND<>   K0 D3410  ; HMI-編輯第11槽電熱設定
      AND<>   K0 D3411  ; HMI-編輯第12槽電熱設定
      AND<>   K0 D3412  ; HMI-編輯進料步進間隔次數設定
      AND<>   K0 D3413  ; HMI-編輯烘烤步進時間設定
      AND<>   K0 D3414  ; HMI-編輯板材尺寸寬度設定
      OUT     M5502  ; 判斷設定參數有效
3719  LDI     M5500  ; 判斷配方ID不為零-1
      ORI     M5501  ; 判斷配方ID不為零-2
      ORI     M5502  ; 判斷設定參數有效
      AND     M5510  ; HMI-PB  配方寫入
      MOV     K1 D5509
3725  LD<>    D5509 K0
      OUT     T1509 K20
      AND     T1509
      MOV     K0 D5509
3735  LD      M5500  ; 判斷配方ID不為零-1
      AND     M5501  ; 判斷配方ID不為零-2
      AND     M5502  ; 判斷設定參數有效
      AND     M5510  ; HMI-PB  配方寫入
      OUT     T1510 K3
      AND     T1510
      SET     M5511  ; 配方寫入-KP
3745  LD      M5511  ; 配方寫入-KP
      MPS
      ANI     T1525
      ANDP    M5512  ; 有相同recipr ID_KP
      RST     M5511  ; 配方寫入-KP
      MRD
      ANI     M5512  ; 有相同recipr ID_KP
      OUT     T1525 K30
      OUT     T1526 K35
      MPP
      MOVP    K1 D5510
      AND     T1526
      RST     M5511  ; 配方寫入-KP
3767  LDI     M5511  ; 配方寫入-KP
      OR<>    D0 K811  ; 人機現在畫頁
      MOV     K0 D5510
3773  LD=     D0 K811  ; 人機現在畫頁
      AND=    K1 D5511
      OUT     T1528 K25
3783  LD      T1528
      OR<>    D0 K811  ; 人機現在畫頁
      MOV     K0 D5511
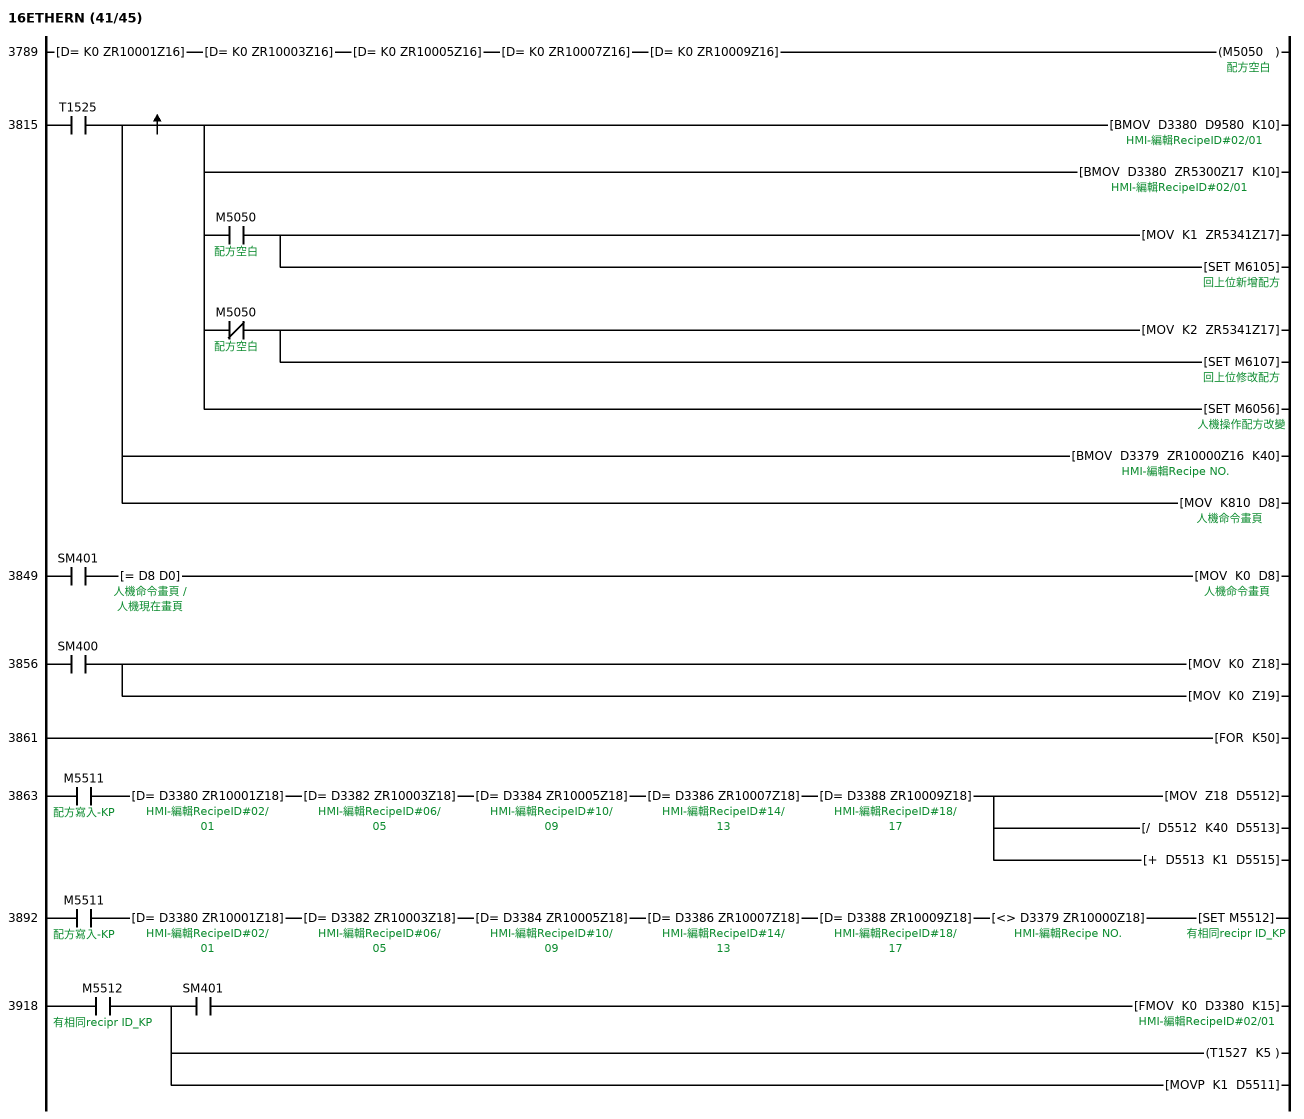
3789  LDD=    K0 ZR10001Z16
      ANDD=   K0 ZR10003Z16
      ANDD=   K0 ZR10005Z16
      ANDD=   K0 ZR10007Z16
      ANDD=   K0 ZR10009Z16
      OUT     M5050  ; 配方空白
3815  LD      T1525
      MPS
      MEP
      BMOV    D3380 D9580 K10
      BMOV    D3380 ZR5300Z17 K10
      MPS
      AND     M5050  ; 配方空白
      MOV     K1 ZR5341Z17
      SET     M6105  ; 回上位新增配方
      MRD
      ANI     M5050  ; 配方空白
      MOV     K2 ZR5341Z17
      SET     M6107  ; 回上位修改配方
      MPP
      SET     M6056  ; 人機操作配方改變
      MPP
      BMOV    D3379 ZR10000Z16 K40
      MOV     K810 D8
3849  LD      SM401
      AND=    D8 D0  ; 人機命令畫頁 / 人機現在畫頁
      MOV     K0 D8
3856  LD      SM400
      MOV     K0 Z18
      MOV     K0 Z19
3861  FOR     K50
3863  LD      M5511  ; 配方寫入-KP
      ANDD=   D3380 ZR10001Z18  ; HMI-編輯RecipeID#02/01
      ANDD=   D3382 ZR10003Z18  ; HMI-編輯RecipeID#06/05
      ANDD=   D3384 ZR10005Z18  ; HMI-編輯RecipeID#10/09
      ANDD=   D3386 ZR10007Z18  ; HMI-編輯RecipeID#14/13
      ANDD=   D3388 ZR10009Z18  ; HMI-編輯RecipeID#18/17
      MOV     Z18 D5512
      /       D5512 K40 D5513
      +       D5513 K1 D5515
3892  LD      M5511  ; 配方寫入-KP
      ANDD=   D3380 ZR10001Z18  ; HMI-編輯RecipeID#02/01
      ANDD=   D3382 ZR10003Z18  ; HMI-編輯RecipeID#06/05
      ANDD=   D3384 ZR10005Z18  ; HMI-編輯RecipeID#10/09
      ANDD=   D3386 ZR10007Z18  ; HMI-編輯RecipeID#14/13
      ANDD=   D3388 ZR10009Z18  ; HMI-編輯RecipeID#18/17
      AND<>   D3379 ZR10000Z18  ; HMI-編輯Recipe NO.
      SET     M5512  ; 有相同recipr ID_KP
3918  LD      M5512  ; 有相同recipr ID_KP
      MPS
      AND     SM401
      FMOV    K0 D3380 K15
      MPP
      OUT     T1527 K5
      MOVP    K1 D5511
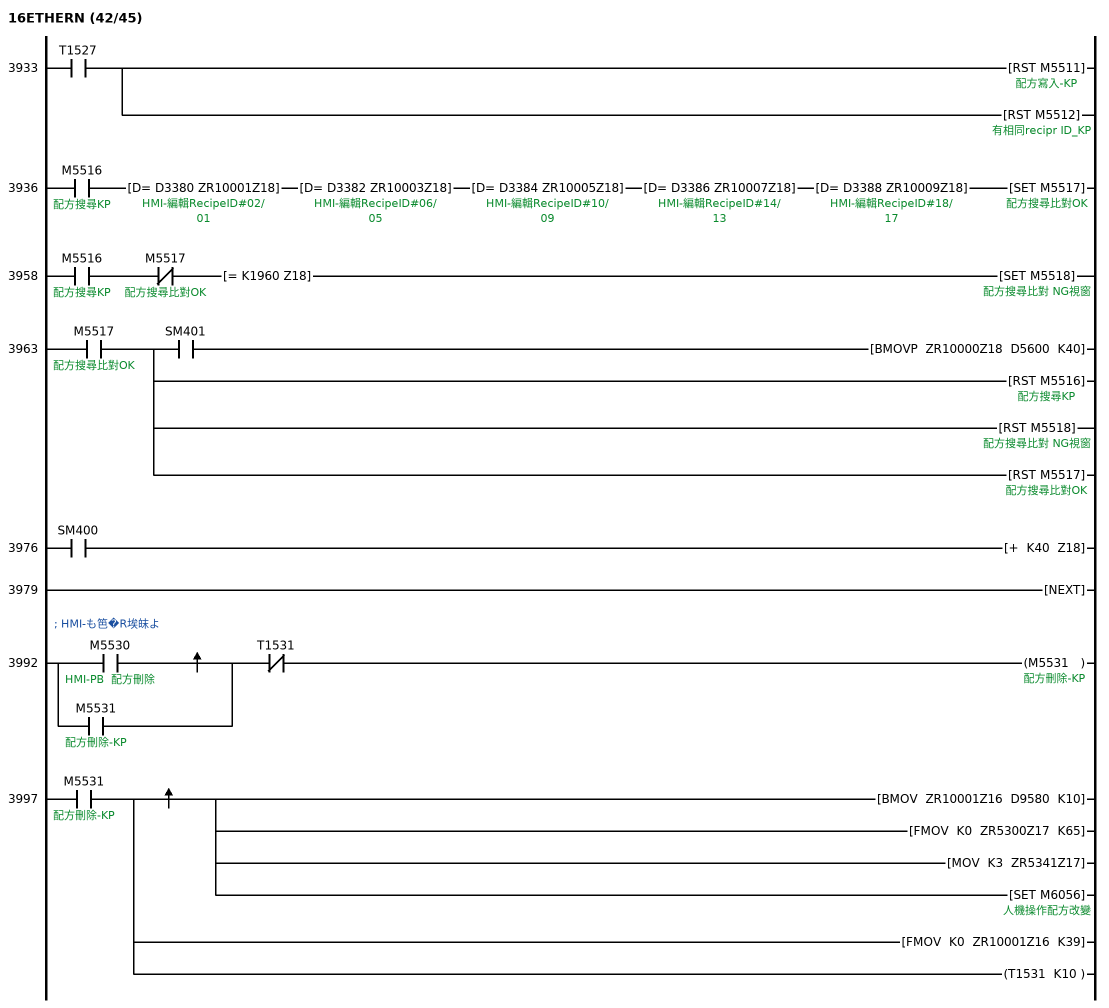
3933  LD      T1527
      RST     M5511  ; 配方寫入-KP
      RST     M5512  ; 有相同recipr ID_KP
3936  LD      M5516  ; 配方搜尋KP
      ANDD=   D3380 ZR10001Z18  ; HMI-編輯RecipeID#02/01
      ANDD=   D3382 ZR10003Z18  ; HMI-編輯RecipeID#06/05
      ANDD=   D3384 ZR10005Z18  ; HMI-編輯RecipeID#10/09
      ANDD=   D3386 ZR10007Z18  ; HMI-編輯RecipeID#14/13
      ANDD=   D3388 ZR10009Z18  ; HMI-編輯RecipeID#18/17
      SET     M5517  ; 配方搜尋比對OK
3958  LD      M5516  ; 配方搜尋KP
      ANI     M5517  ; 配方搜尋比對OK
      AND=    K1960 Z18
      SET     M5518  ; 配方搜尋比對 NG視窗
3963  LD      M5517  ; 配方搜尋比對OK
      MPS
      AND     SM401
      BMOVP   ZR10000Z18 D5600 K40
      MPP
      RST     M5516  ; 配方搜尋KP
      RST     M5518  ; 配方搜尋比對 NG視窗
      RST     M5517  ; 配方搜尋比對OK
3976  LD      SM400
      +       K40 Z18
3979  NEXT
; HMI-手動刪除配方
3992  LD      M5530  ; HMI-PB  配方刪除
      MEP
      OR      M5531  ; 配方刪除-KP
      ANI     T1531
      OUT     M5531  ; 配方刪除-KP
3997  LD      M5531  ; 配方刪除-KP
      MPS
      MEP
      BMOV    ZR10001Z16 D9580 K10
      FMOV    K0 ZR5300Z17 K65
      MOV     K3 ZR5341Z17
      SET     M6056  ; 人機操作配方改變
      MPP
      FMOV    K0 ZR10001Z16 K39
      OUT     T1531 K10
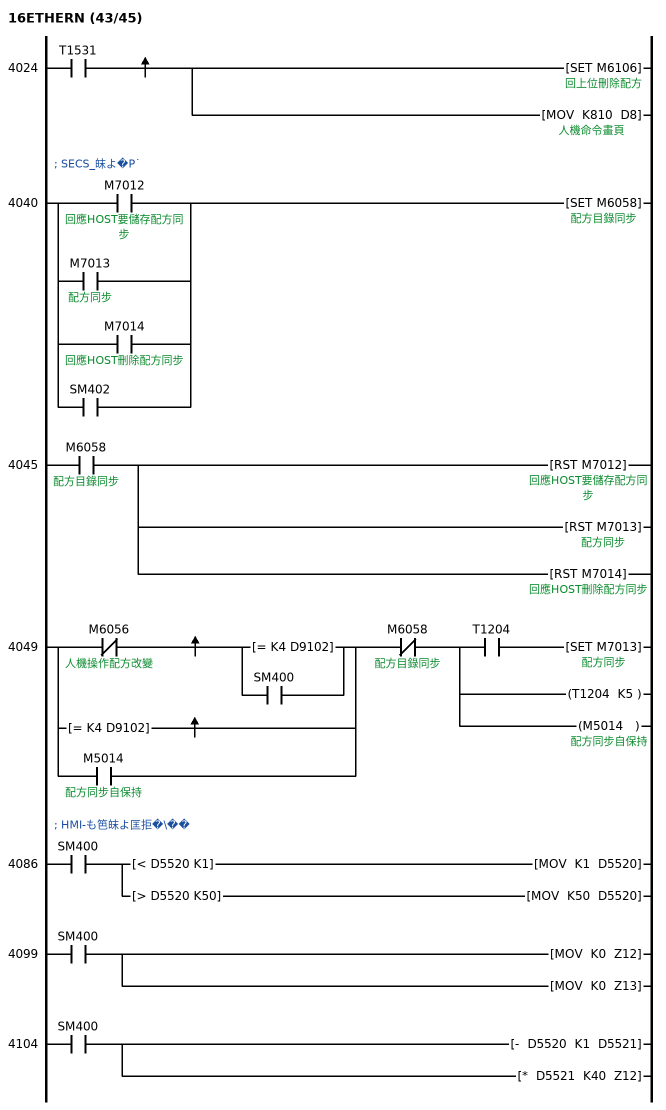
4024  LD      T1531
      MEP
      SET     M6106  ; 回上位刪除配方
      MOV     K810 D8
; SECS_配方同步
4040  LD      M7012  ; 回應HOST要儲存配方同步
      OR      M7013  ; 配方同步
      OR      M7014  ; 回應HOST刪除配方同步
      OR      SM402
      SET     M6058  ; 配方目錄同步
4045  LD      M6058  ; 配方目錄同步
      RST     M7012  ; 回應HOST要儲存配方同步
      RST     M7013  ; 配方同步
      RST     M7014  ; 回應HOST刪除配方同步
4049  LDI     M6056  ; 人機操作配方改變
      MEP
      LD=     K4 D9102
      OR      SM400
      ANB
      LD=     K4 D9102
      MEP
      ORB
      OR      M5014  ; 配方同步自保持
      ANI     M6058  ; 配方目錄同步
      MPS
      AND     T1204
      SET     M7013  ; 配方同步
      MPP
      OUT     T1204 K5
      OUT     M5014  ; 配方同步自保持
; HMI-手動配方選擇功能
4086  LD      SM400
      MPS
      AND<    D5520 K1
      MOV     K1 D5520
      MPP
      AND>    D5520 K50
      MOV     K50 D5520
4099  LD      SM400
      MOV     K0 Z12
      MOV     K0 Z13
4104  LD      SM400
      -       D5520 K1 D5521
      *       D5521 K40 Z12
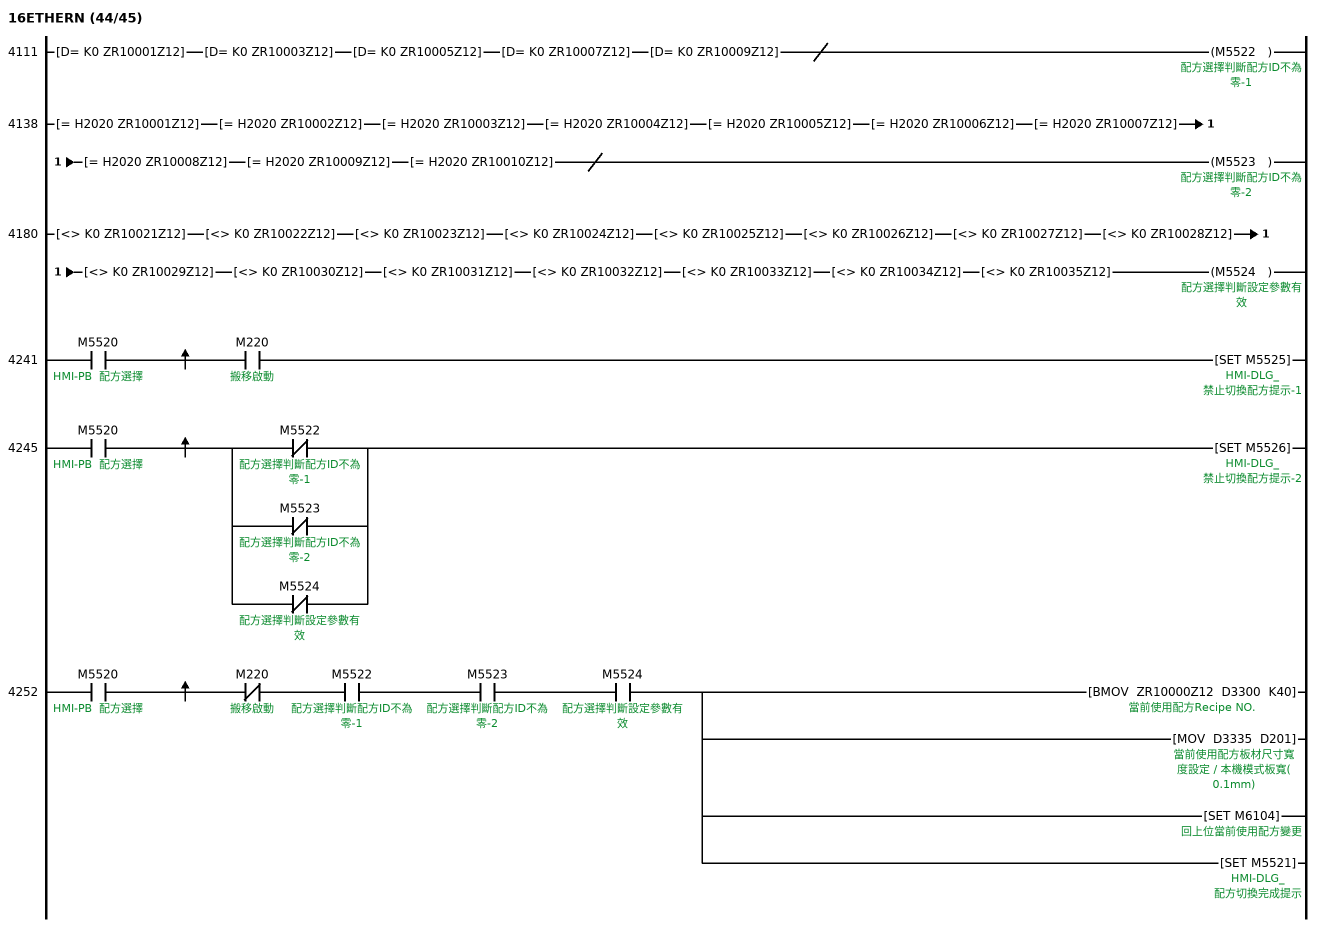
4111  LDD=    K0 ZR10001Z12
      ANDD=   K0 ZR10003Z12
      ANDD=   K0 ZR10005Z12
      ANDD=   K0 ZR10007Z12
      ANDD=   K0 ZR10009Z12
      INV
      OUT     M5522  ; 配方選擇判斷配方ID不為零-1
4138  LD=     H2020 ZR10001Z12
      AND=    H2020 ZR10002Z12
      AND=    H2020 ZR10003Z12
      AND=    H2020 ZR10004Z12
      AND=    H2020 ZR10005Z12
      AND=    H2020 ZR10006Z12
      AND=    H2020 ZR10007Z12
      AND=    H2020 ZR10008Z12
      AND=    H2020 ZR10009Z12
      AND=    H2020 ZR10010Z12
      INV
      OUT     M5523  ; 配方選擇判斷配方ID不為零-2
4180  LD<>    K0 ZR10021Z12
      AND<>   K0 ZR10022Z12
      AND<>   K0 ZR10023Z12
      AND<>   K0 ZR10024Z12
      AND<>   K0 ZR10025Z12
      AND<>   K0 ZR10026Z12
      AND<>   K0 ZR10027Z12
      AND<>   K0 ZR10028Z12
      AND<>   K0 ZR10029Z12
      AND<>   K0 ZR10030Z12
      AND<>   K0 ZR10031Z12
      AND<>   K0 ZR10032Z12
      AND<>   K0 ZR10033Z12
      AND<>   K0 ZR10034Z12
      AND<>   K0 ZR10035Z12
      OUT     M5524  ; 配方選擇判斷設定參數有效
4241  LD      M5520  ; HMI-PB  配方選擇
      MEP
      AND     M220  ; 搬移啟動
      SET     M5525  ; HMI-DLG_禁止切換配方提示-1
4245  LD      M5520  ; HMI-PB  配方選擇
      MEP
      LDI     M5522  ; 配方選擇判斷配方ID不為零-1
      ORI     M5523  ; 配方選擇判斷配方ID不為零-2
      ORI     M5524  ; 配方選擇判斷設定參數有效
      ANB
      SET     M5526  ; HMI-DLG_禁止切換配方提示-2
4252  LD      M5520  ; HMI-PB  配方選擇
      MEP
      ANI     M220  ; 搬移啟動
      AND     M5522  ; 配方選擇判斷配方ID不為零-1
      AND     M5523  ; 配方選擇判斷配方ID不為零-2
      AND     M5524  ; 配方選擇判斷設定參數有效
      BMOV    ZR10000Z12 D3300 K40
      MOV     D3335 D201
      SET     M6104  ; 回上位當前使用配方變更
      SET     M5521  ; HMI-DLG_配方切換完成提示
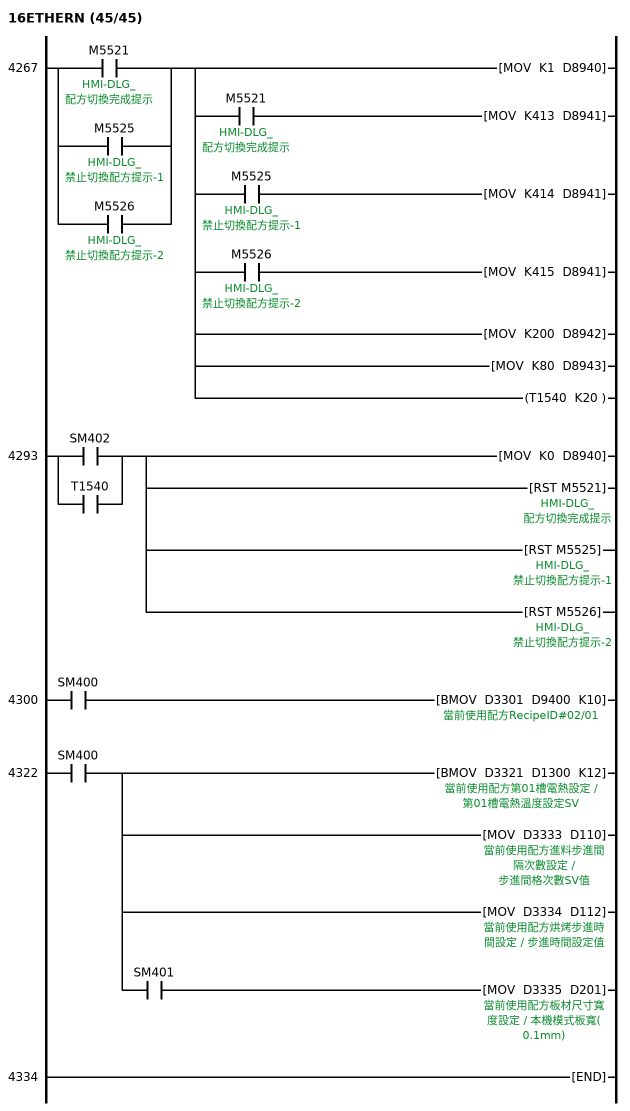
4267  LD      M5521  ; HMI-DLG_配方切換完成提示
      OR      M5525  ; HMI-DLG_禁止切換配方提示-1
      OR      M5526  ; HMI-DLG_禁止切換配方提示-2
      MOV     K1 D8940
      MPS
      AND     M5521  ; HMI-DLG_配方切換完成提示
      MOV     K413 D8941
      MRD
      AND     M5525  ; HMI-DLG_禁止切換配方提示-1
      MOV     K414 D8941
      MRD
      AND     M5526  ; HMI-DLG_禁止切換配方提示-2
      MOV     K415 D8941
      MPP
      MOV     K200 D8942
      MOV     K80 D8943
      OUT     T1540 K20
4293  LD      SM402
      OR      T1540
      MOV     K0 D8940
      RST     M5521  ; HMI-DLG_配方切換完成提示
      RST     M5525  ; HMI-DLG_禁止切換配方提示-1
      RST     M5526  ; HMI-DLG_禁止切換配方提示-2
4300  LD      SM400
      BMOV    D3301 D9400 K10  ; 當前使用配方RecipeID#02/01
        [note] D9400_上報SECS目前使用PPID名稱
4322  LD      SM400
      BMOV    D3321 D1300 K12  ; 當前使用配方第01槽電熱設定
      MOV     D3333 D110  ; 當前使用配方進料步進間隔次數設定
      MOV     D3334 D112  ; 當前使用配方烘烤步進時間設定
      AND     SM401
      MOV     D3335 D201
4334  END
END_PROGRAM

PROGRAM 17GBF-20
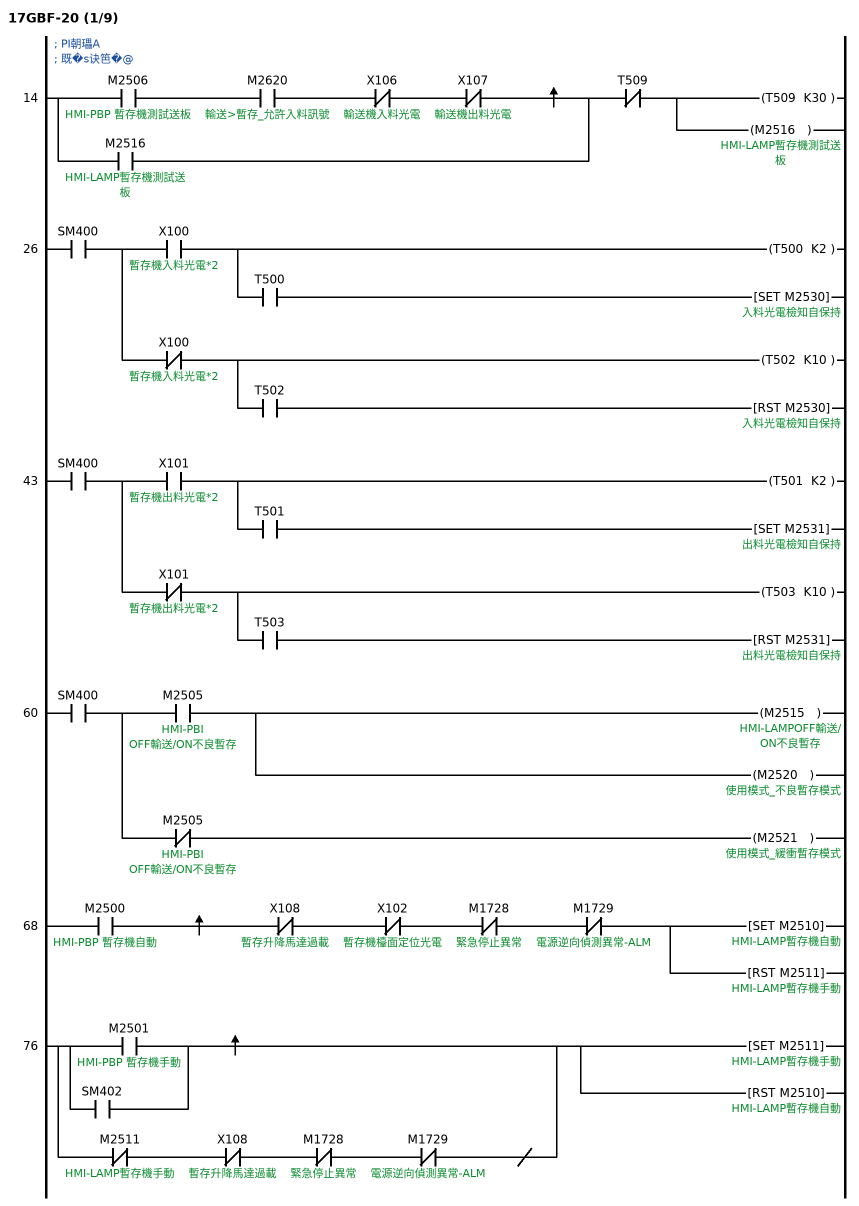
; PI朝瓃Α
; 暫存機動作
14    LD      M2506  ; HMI-PBP 暫存機測試送板
      AND     M2620  ; 輸送>暫存_允許入料訊號
      ANI     X106  ; 輸送機入料光電
      ANI     X107  ; 輸送機出料光電
      MEP
      OR      M2516  ; HMI-LAMP暫存機測試送板
      ANI     T509
      OUT     T509 K30
      OUT     M2516  ; HMI-LAMP暫存機測試送板
26    LD      SM400
      MPS
      AND     X100  ; 暫存機入料光電*2
      OUT     T500 K2
      AND     T500
      SET     M2530  ; 入料光電檢知自保持
      MPP
      ANI     X100  ; 暫存機入料光電*2
      OUT     T502 K10
      AND     T502
      RST     M2530  ; 入料光電檢知自保持
43    LD      SM400
      MPS
      AND     X101  ; 暫存機出料光電*2
      OUT     T501 K2
      AND     T501
      SET     M2531  ; 出料光電檢知自保持
      MPP
      ANI     X101  ; 暫存機出料光電*2
      OUT     T503 K10
      AND     T503
      RST     M2531  ; 出料光電檢知自保持
60    LD      SM400
      MPS
      AND     M2505  ; HMI-PBI OFF輸送/ON不良暫存
      OUT     M2515  ; HMI-LAMPOFF輸送/ON不良暫存
      OUT     M2520  ; 使用模式_不良暫存模式
      MPP
      ANI     M2505  ; HMI-PBI OFF輸送/ON不良暫存
      OUT     M2521  ; 使用模式_緩衝暫存模式
68    LD      M2500  ; HMI-PBP 暫存機自動
      MEP
      ANI     X108  ; 暫存升降馬達過載
      ANI     X102  ; 暫存機檯面定位光電
      ANI     M1728  ; 緊急停止異常
      ANI     M1729  ; 電源逆向偵測異常-ALM
      SET     M2510  ; HMI-LAMP暫存機自動
      RST     M2511  ; HMI-LAMP暫存機手動
76    LD      M2501  ; HMI-PBP 暫存機手動
      OR      SM402
      MEP
      LDI     M2511  ; HMI-LAMP暫存機手動
      ANI     X108  ; 暫存升降馬達過載
      ANI     M1728  ; 緊急停止異常
      ANI     M1729  ; 電源逆向偵測異常-ALM
      INV
      ORB
      SET     M2511  ; HMI-LAMP暫存機手動
      RST     M2510  ; HMI-LAMP暫存機自動
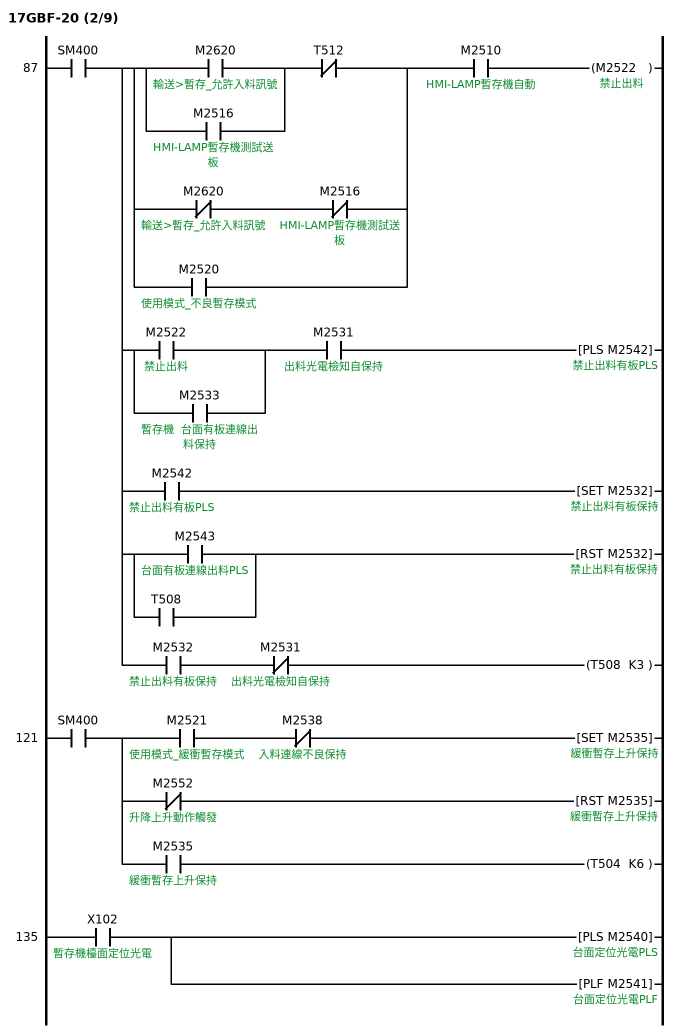
87    LD      SM400
      MPS
      LD      M2620  ; 輸送>暫存_允許入料訊號
      OR      M2516  ; HMI-LAMP暫存機測試送板
      ANI     T512
      LDI     M2620  ; 輸送>暫存_允許入料訊號
      ANI     M2516  ; HMI-LAMP暫存機測試送板
      ORB
      OR      M2520  ; 使用模式_不良暫存模式
      ANB
      AND     M2510  ; HMI-LAMP暫存機自動
      OUT     M2522  ; 禁止出料
      MRD
      LD      M2522  ; 禁止出料
      OR      M2533  ; 暫存機  台面有板連線出料保持
      ANB
      AND     M2531  ; 出料光電檢知自保持
      PLS     M2542  ; 禁止出料有板PLS
      MRD
      AND     M2542  ; 禁止出料有板PLS
      SET     M2532  ; 禁止出料有板保持
      MRD
      LD      M2543  ; 台面有板連線出料PLS
      OR      T508
      ANB
      RST     M2532  ; 禁止出料有板保持
      MPP
      AND     M2532  ; 禁止出料有板保持
      ANI     M2531  ; 出料光電檢知自保持
      OUT     T508 K3
121   LD      SM400
      MPS
      AND     M2521  ; 使用模式_緩衝暫存模式
      ANI     M2538  ; 入料連線不良保持
      SET     M2535  ; 緩衝暫存上升保持
      MRD
      ANI     M2552  ; 升降上升動作觸發
      RST     M2535  ; 緩衝暫存上升保持
      MPP
      AND     M2535  ; 緩衝暫存上升保持
      OUT     T504 K6
135   LD      X102  ; 暫存機檯面定位光電
      PLS     M2540  ; 台面定位光電PLS
      PLF     M2541  ; 台面定位光電PLF
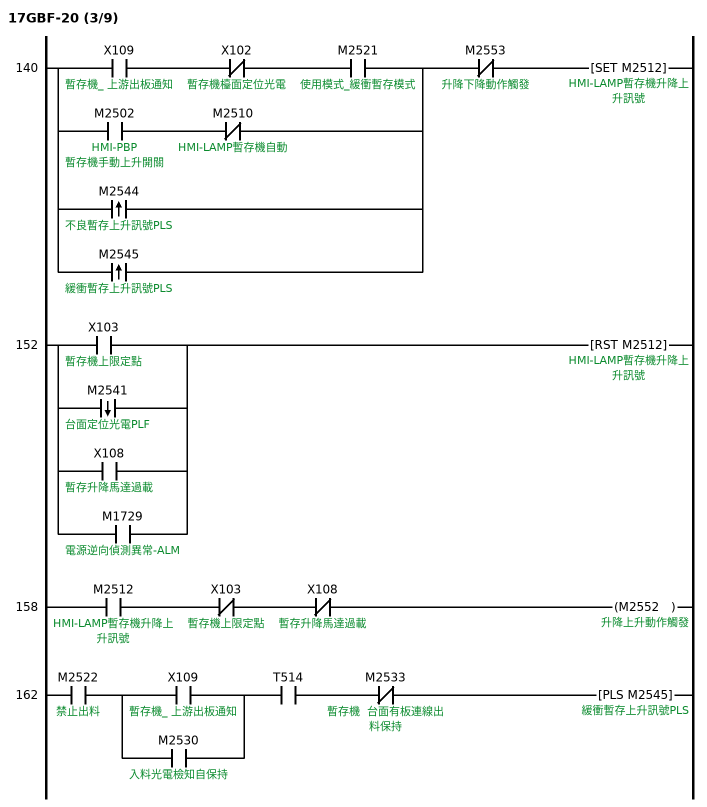
140   LD      X109  ; 暫存機_ 上游出板通知
      ANI     X102  ; 暫存機檯面定位光電
      AND     M2521  ; 使用模式_緩衝暫存模式
      LD      M2502  ; HMI-PBP 暫存機手動上升開關
      ANI     M2510  ; HMI-LAMP暫存機自動
      ORB
      ORP     M2544  ; 不良暫存上升訊號PLS
      ORP     M2545  ; 緩衝暫存上升訊號PLS
      ANI     M2553  ; 升降下降動作觸發
      SET     M2512  ; HMI-LAMP暫存機升降上升訊號
152   LD      X103  ; 暫存機上限定點
      ORF     M2541  ; 台面定位光電PLF
      OR      X108  ; 暫存升降馬達過載
      OR      M1729  ; 電源逆向偵測異常-ALM
      RST     M2512  ; HMI-LAMP暫存機升降上升訊號
158   LD      M2512  ; HMI-LAMP暫存機升降上升訊號
      ANI     X103  ; 暫存機上限定點
      ANI     X108  ; 暫存升降馬達過載
      OUT     M2552  ; 升降上升動作觸發
162   LD      M2522  ; 禁止出料
      LD      X109  ; 暫存機_ 上游出板通知
      OR      M2530  ; 入料光電檢知自保持
      ANB
      AND     T514
      ANI     M2533  ; 暫存機  台面有板連線出料保持
      PLS     M2545  ; 緩衝暫存上升訊號PLS
